REGION Network 3: Обработка аварии по входу №0 / Input 0
   LAB1:
   IF #Input_0 THEN
       #Tmp_Real := #Delay_Sec_0 * 1000.0;
       #Tmp_Time := ROUND(#Tmp_Real);
   END_IF;
   #Timer_0(IN := #Input_0, PT := #Tmp_Time);   // TON
   #_w1 := #Timer_0.Q AND NOT #sarxArrayFlanke[0];   // rising edge
   #sarxArrayFlanke[0] := #Timer_0.Q;
   #sarxArrayMerkers[0] := #_w1;
   #Alarm_0 := (NOT #sarxArrayMerkers[0] AND #Alarm_0) OR (#sarxArrayMerkers[0] AND NOT #Alarm_0);
END_REGION

REGION Network 4: Обработка аварии по входу №1 / Input 1
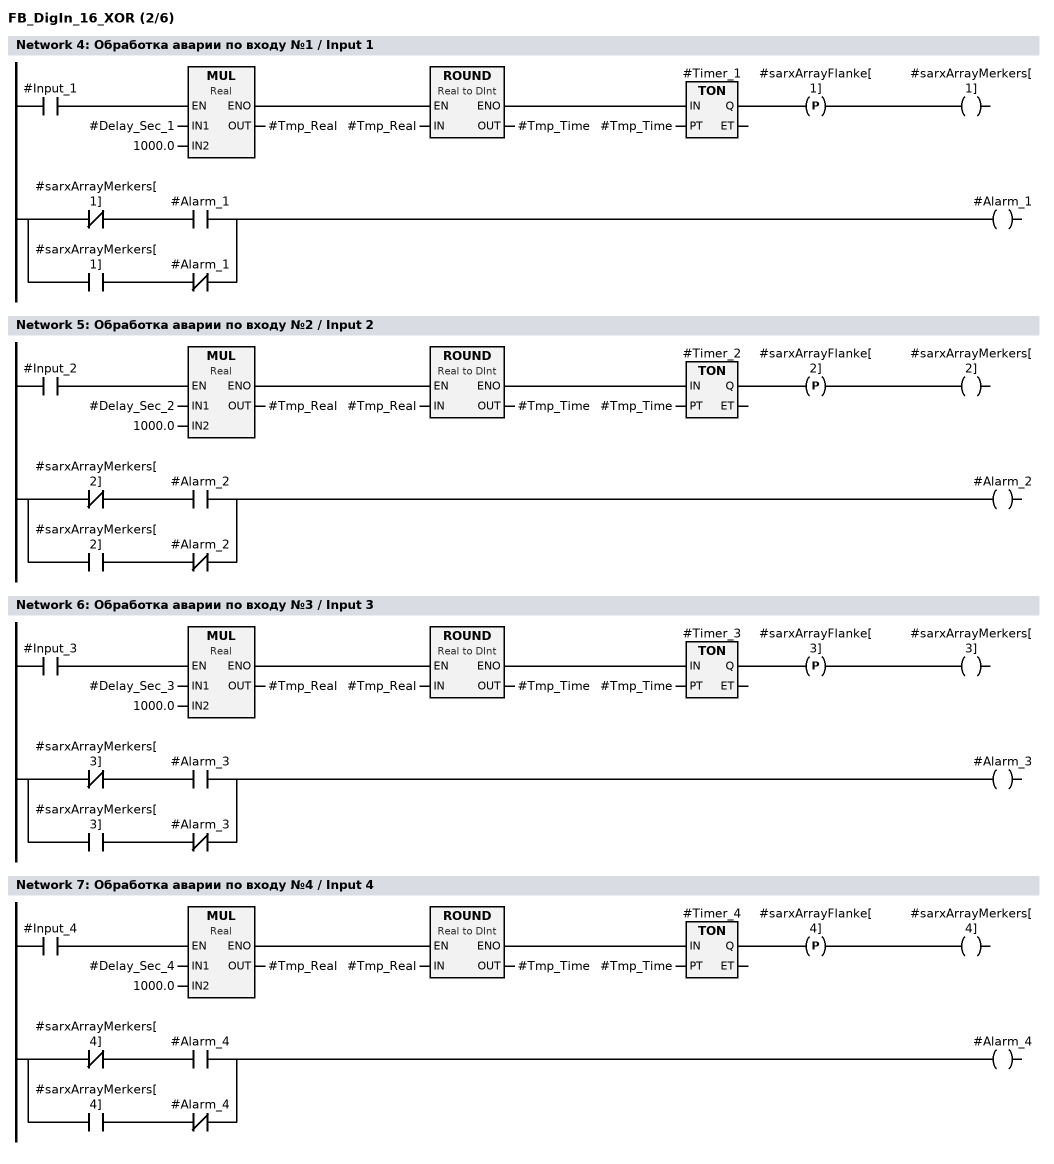
   IF #Input_1 THEN
       #Tmp_Real := #Delay_Sec_1 * 1000.0;
       #Tmp_Time := ROUND(#Tmp_Real);
   END_IF;
   #Timer_1(IN := #Input_1, PT := #Tmp_Time);   // TON
   #_w1 := #Timer_1.Q AND NOT #sarxArrayFlanke[1];   // rising edge
   #sarxArrayFlanke[1] := #Timer_1.Q;
   #sarxArrayMerkers[1] := #_w1;
   #Alarm_1 := (NOT #sarxArrayMerkers[1] AND #Alarm_1) OR (#sarxArrayMerkers[1] AND NOT #Alarm_1);
END_REGION

REGION Network 5: Обработка аварии по входу №2 / Input 2
   IF #Input_2 THEN
       #Tmp_Real := #Delay_Sec_2 * 1000.0;
       #Tmp_Time := ROUND(#Tmp_Real);
   END_IF;
   #Timer_2(IN := #Input_2, PT := #Tmp_Time);   // TON
   #_w1 := #Timer_2.Q AND NOT #sarxArrayFlanke[2];   // rising edge
   #sarxArrayFlanke[2] := #Timer_2.Q;
   #sarxArrayMerkers[2] := #_w1;
   #Alarm_2 := (NOT #sarxArrayMerkers[2] AND #Alarm_2) OR (#sarxArrayMerkers[2] AND NOT #Alarm_2);
END_REGION

REGION Network 6: Обработка аварии по входу №3 / Input 3
   IF #Input_3 THEN
       #Tmp_Real := #Delay_Sec_3 * 1000.0;
       #Tmp_Time := ROUND(#Tmp_Real);
   END_IF;
   #Timer_3(IN := #Input_3, PT := #Tmp_Time);   // TON
   #_w1 := #Timer_3.Q AND NOT #sarxArrayFlanke[3];   // rising edge
   #sarxArrayFlanke[3] := #Timer_3.Q;
   #sarxArrayMerkers[3] := #_w1;
   #Alarm_3 := (NOT #sarxArrayMerkers[3] AND #Alarm_3) OR (#sarxArrayMerkers[3] AND NOT #Alarm_3);
END_REGION

REGION Network 7: Обработка аварии по входу №4 / Input 4
   IF #Input_4 THEN
       #Tmp_Real := #Delay_Sec_4 * 1000.0;
       #Tmp_Time := ROUND(#Tmp_Real);
   END_IF;
   #Timer_4(IN := #Input_4, PT := #Tmp_Time);   // TON
   #_w1 := #Timer_4.Q AND NOT #sarxArrayFlanke[4];   // rising edge
   #sarxArrayFlanke[4] := #Timer_4.Q;
   #sarxArrayMerkers[4] := #_w1;
   #Alarm_4 := (NOT #sarxArrayMerkers[4] AND #Alarm_4) OR (#sarxArrayMerkers[4] AND NOT #Alarm_4);
END_REGION

REGION Network 8: Обработка аварии по входу №5 / Input 5
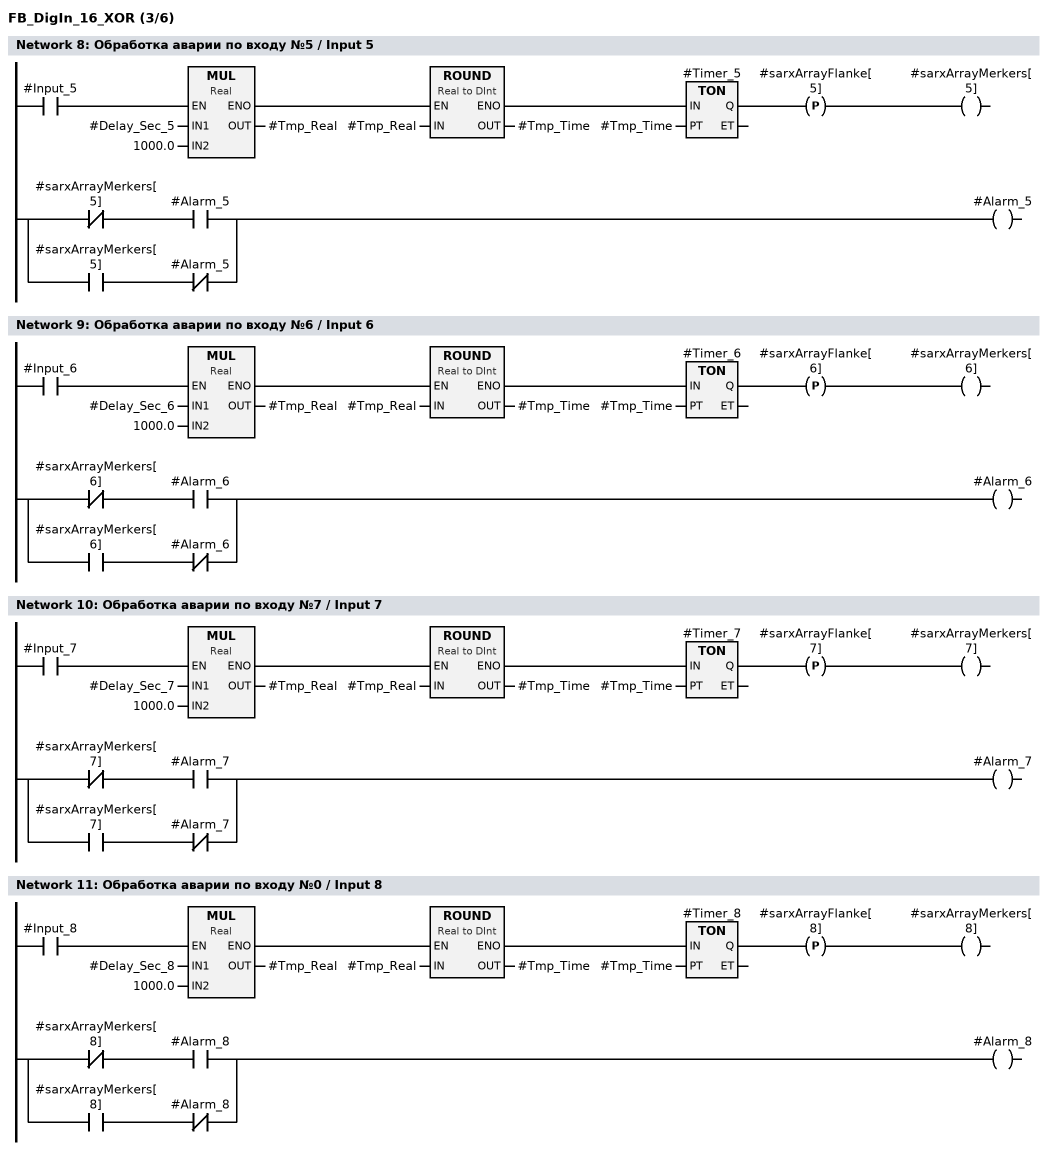
   IF #Input_5 THEN
       #Tmp_Real := #Delay_Sec_5 * 1000.0;
       #Tmp_Time := ROUND(#Tmp_Real);
   END_IF;
   #Timer_5(IN := #Input_5, PT := #Tmp_Time);   // TON
   #_w1 := #Timer_5.Q AND NOT #sarxArrayFlanke[5];   // rising edge
   #sarxArrayFlanke[5] := #Timer_5.Q;
   #sarxArrayMerkers[5] := #_w1;
   #Alarm_5 := (NOT #sarxArrayMerkers[5] AND #Alarm_5) OR (#sarxArrayMerkers[5] AND NOT #Alarm_5);
END_REGION

REGION Network 9: Обработка аварии по входу №6 / Input 6
   IF #Input_6 THEN
       #Tmp_Real := #Delay_Sec_6 * 1000.0;
       #Tmp_Time := ROUND(#Tmp_Real);
   END_IF;
   #Timer_6(IN := #Input_6, PT := #Tmp_Time);   // TON
   #_w1 := #Timer_6.Q AND NOT #sarxArrayFlanke[6];   // rising edge
   #sarxArrayFlanke[6] := #Timer_6.Q;
   #sarxArrayMerkers[6] := #_w1;
   #Alarm_6 := (NOT #sarxArrayMerkers[6] AND #Alarm_6) OR (#sarxArrayMerkers[6] AND NOT #Alarm_6);
END_REGION

REGION Network 10: Обработка аварии по входу №7 / Input 7
   IF #Input_7 THEN
       #Tmp_Real := #Delay_Sec_7 * 1000.0;
       #Tmp_Time := ROUND(#Tmp_Real);
   END_IF;
   #Timer_7(IN := #Input_7, PT := #Tmp_Time);   // TON
   #_w1 := #Timer_7.Q AND NOT #sarxArrayFlanke[7];   // rising edge
   #sarxArrayFlanke[7] := #Timer_7.Q;
   #sarxArrayMerkers[7] := #_w1;
   #Alarm_7 := (NOT #sarxArrayMerkers[7] AND #Alarm_7) OR (#sarxArrayMerkers[7] AND NOT #Alarm_7);
END_REGION

REGION Network 11: Обработка аварии по входу №0 / Input 8
   IF #Input_8 THEN
       #Tmp_Real := #Delay_Sec_8 * 1000.0;
       #Tmp_Time := ROUND(#Tmp_Real);
   END_IF;
   #Timer_8(IN := #Input_8, PT := #Tmp_Time);   // TON
   #_w1 := #Timer_8.Q AND NOT #sarxArrayFlanke[8];   // rising edge
   #sarxArrayFlanke[8] := #Timer_8.Q;
   #sarxArrayMerkers[8] := #_w1;
   #Alarm_8 := (NOT #sarxArrayMerkers[8] AND #Alarm_8) OR (#sarxArrayMerkers[8] AND NOT #Alarm_8);
END_REGION

REGION Network 12: Обработка аварии по входу №0 / Input 9
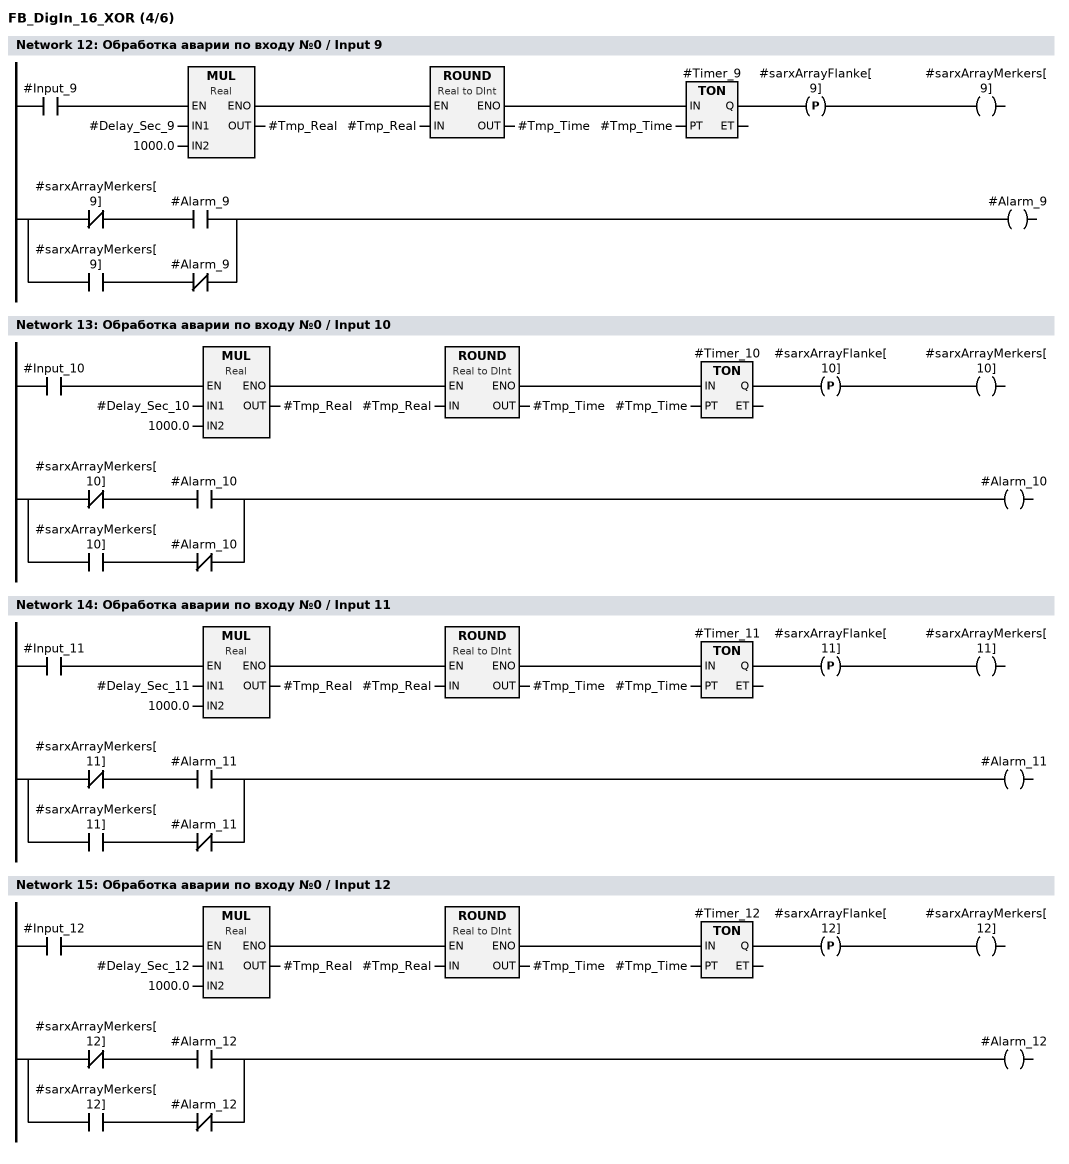
   IF #Input_9 THEN
       #Tmp_Real := #Delay_Sec_9 * 1000.0;
       #Tmp_Time := ROUND(#Tmp_Real);
   END_IF;
   #Timer_9(IN := #Input_9, PT := #Tmp_Time);   // TON
   #_w1 := #Timer_9.Q AND NOT #sarxArrayFlanke[9];   // rising edge
   #sarxArrayFlanke[9] := #Timer_9.Q;
   #sarxArrayMerkers[9] := #_w1;
   #Alarm_9 := (NOT #sarxArrayMerkers[9] AND #Alarm_9) OR (#sarxArrayMerkers[9] AND NOT #Alarm_9);
END_REGION

REGION Network 13: Обработка аварии по входу №0 / Input 10
   IF #Input_10 THEN
       #Tmp_Real := #Delay_Sec_10 * 1000.0;
       #Tmp_Time := ROUND(#Tmp_Real);
   END_IF;
   #Timer_10(IN := #Input_10, PT := #Tmp_Time);   // TON
   #_w1 := #Timer_10.Q AND NOT #sarxArrayFlanke[10];   // rising edge
   #sarxArrayFlanke[10] := #Timer_10.Q;
   #sarxArrayMerkers[10] := #_w1;
   #Alarm_10 := (NOT #sarxArrayMerkers[10] AND #Alarm_10) OR (#sarxArrayMerkers[10] AND NOT #Alarm_10);
END_REGION

REGION Network 14: Обработка аварии по входу №0 / Input 11
   IF #Input_11 THEN
       #Tmp_Real := #Delay_Sec_11 * 1000.0;
       #Tmp_Time := ROUND(#Tmp_Real);
   END_IF;
   #Timer_11(IN := #Input_11, PT := #Tmp_Time);   // TON
   #_w1 := #Timer_11.Q AND NOT #sarxArrayFlanke[11];   // rising edge
   #sarxArrayFlanke[11] := #Timer_11.Q;
   #sarxArrayMerkers[11] := #_w1;
   #Alarm_11 := (NOT #sarxArrayMerkers[11] AND #Alarm_11) OR (#sarxArrayMerkers[11] AND NOT #Alarm_11);
END_REGION

REGION Network 15: Обработка аварии по входу №0 / Input 12
   IF #Input_12 THEN
       #Tmp_Real := #Delay_Sec_12 * 1000.0;
       #Tmp_Time := ROUND(#Tmp_Real);
   END_IF;
   #Timer_12(IN := #Input_12, PT := #Tmp_Time);   // TON
   #_w1 := #Timer_12.Q AND NOT #sarxArrayFlanke[12];   // rising edge
   #sarxArrayFlanke[12] := #Timer_12.Q;
   #sarxArrayMerkers[12] := #_w1;
   #Alarm_12 := (NOT #sarxArrayMerkers[12] AND #Alarm_12) OR (#sarxArrayMerkers[12] AND NOT #Alarm_12);
END_REGION

REGION Network 16: Обработка аварии по входу №0 / Input 13
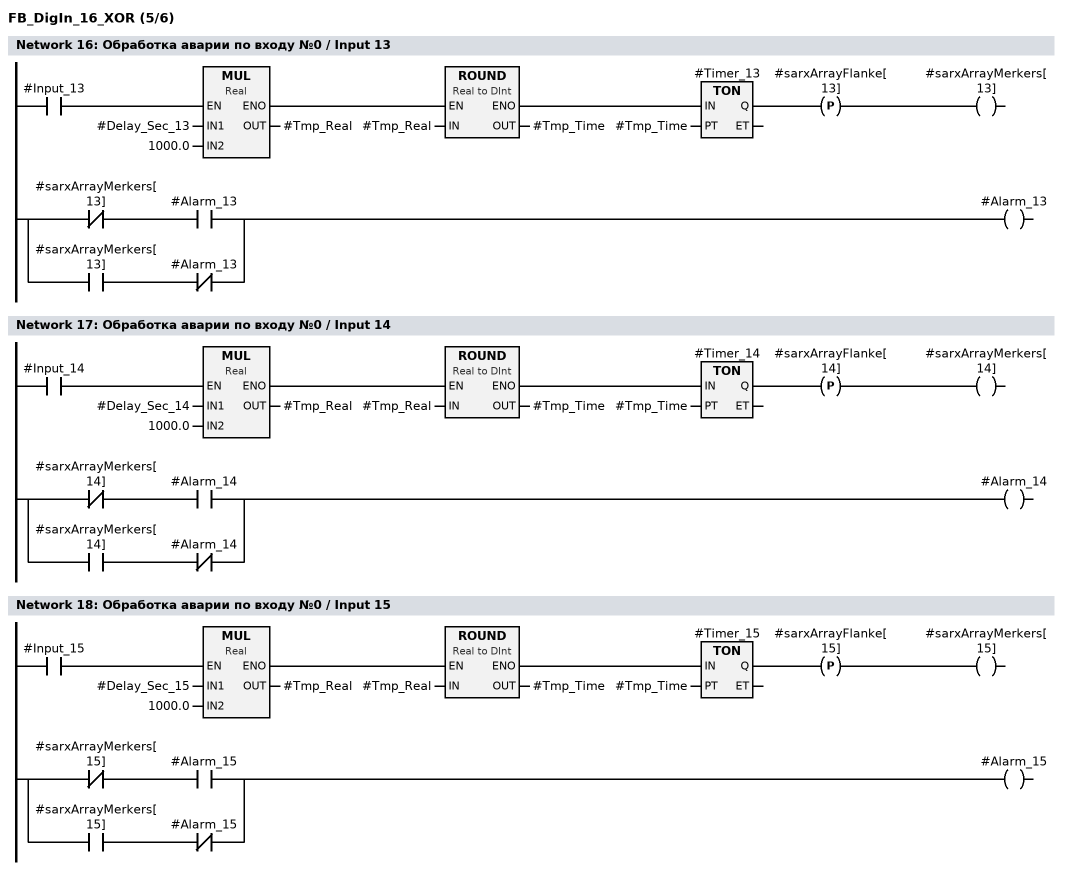
   IF #Input_13 THEN
       #Tmp_Real := #Delay_Sec_13 * 1000.0;
       #Tmp_Time := ROUND(#Tmp_Real);
   END_IF;
   #Timer_13(IN := #Input_13, PT := #Tmp_Time);   // TON
   #_w1 := #Timer_13.Q AND NOT #sarxArrayFlanke[13];   // rising edge
   #sarxArrayFlanke[13] := #Timer_13.Q;
   #sarxArrayMerkers[13] := #_w1;
   #Alarm_13 := (NOT #sarxArrayMerkers[13] AND #Alarm_13) OR (#sarxArrayMerkers[13] AND NOT #Alarm_13);
END_REGION

REGION Network 17: Обработка аварии по входу №0 / Input 14
   IF #Input_14 THEN
       #Tmp_Real := #Delay_Sec_14 * 1000.0;
       #Tmp_Time := ROUND(#Tmp_Real);
   END_IF;
   #Timer_14(IN := #Input_14, PT := #Tmp_Time);   // TON
   #_w1 := #Timer_14.Q AND NOT #sarxArrayFlanke[14];   // rising edge
   #sarxArrayFlanke[14] := #Timer_14.Q;
   #sarxArrayMerkers[14] := #_w1;
   #Alarm_14 := (NOT #sarxArrayMerkers[14] AND #Alarm_14) OR (#sarxArrayMerkers[14] AND NOT #Alarm_14);
END_REGION

REGION Network 18: Обработка аварии по входу №0 / Input 15
   IF #Input_15 THEN
       #Tmp_Real := #Delay_Sec_15 * 1000.0;
       #Tmp_Time := ROUND(#Tmp_Real);
   END_IF;
   #Timer_15(IN := #Input_15, PT := #Tmp_Time);   // TON
   #_w1 := #Timer_15.Q AND NOT #sarxArrayFlanke[15];   // rising edge
   #sarxArrayFlanke[15] := #Timer_15.Q;
   #sarxArrayMerkers[15] := #_w1;
   #Alarm_15 := (NOT #sarxArrayMerkers[15] AND #Alarm_15) OR (#sarxArrayMerkers[15] AND NOT #Alarm_15);
END_REGION

REGION Network 19: Формування статусних слів
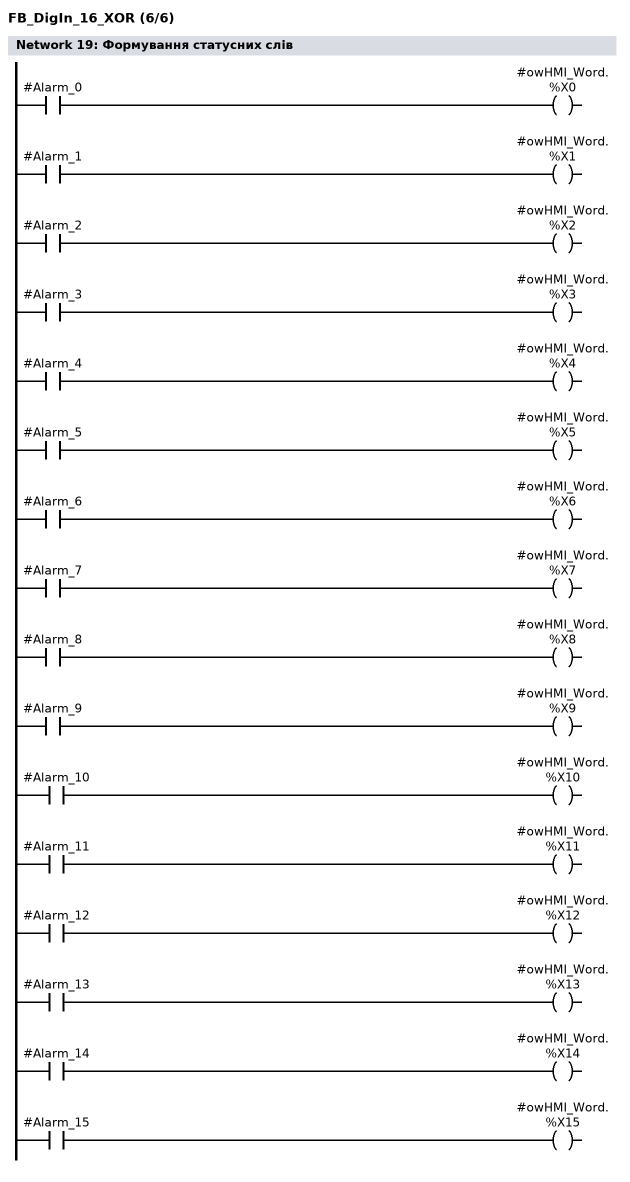
   RUNG wire#powerrail
      Contact( #Alarm_0 )
      Coil( #owHMI_Word.%X0 )
   END_RUNG
   RUNG wire#powerrail
      Contact( #Alarm_1 )
      Coil( #owHMI_Word.%X1 )
   END_RUNG
   RUNG wire#powerrail
      Contact( #Alarm_2 )
      Coil( #owHMI_Word.%X2 )
   END_RUNG
   RUNG wire#powerrail
      Contact( #Alarm_3 )
      Coil( #owHMI_Word.%X3 )
   END_RUNG
   RUNG wire#powerrail
      Contact( #Alarm_4 )
      Coil( #owHMI_Word.%X4 )
   END_RUNG
   RUNG wire#powerrail
      Contact( #Alarm_5 )
      Coil( #owHMI_Word.%X5 )
   END_RUNG
   RUNG wire#powerrail
      Contact( #Alarm_6 )
      Coil( #owHMI_Word.%X6 )
   END_RUNG
   RUNG wire#powerrail
      Contact( #Alarm_7 )
      Coil( #owHMI_Word.%X7 )
   END_RUNG
   RUNG wire#powerrail
      Contact( #Alarm_8 )
      Coil( #owHMI_Word.%X8 )
   END_RUNG
   RUNG wire#powerrail
      Contact( #Alarm_9 )
      Coil( #owHMI_Word.%X9 )
   END_RUNG
   RUNG wire#powerrail
      Contact( #Alarm_10 )
      Coil( #owHMI_Word.%X10 )
   END_RUNG
   RUNG wire#powerrail
      Contact( #Alarm_11 )
      Coil( #owHMI_Word.%X11 )
   END_RUNG
   RUNG wire#powerrail
      Contact( #Alarm_12 )
      Coil( #owHMI_Word.%X12 )
   END_RUNG
   RUNG wire#powerrail
      Contact( #Alarm_13 )
      Coil( #owHMI_Word.%X13 )
   END_RUNG
   RUNG wire#powerrail
      Contact( #Alarm_14 )
      Coil( #owHMI_Word.%X14 )
   END_RUNG
   RUNG wire#powerrail
      Contact( #Alarm_15 )
      Coil( #owHMI_Word.%X15 )
   END_RUNG
   // the same network as SCL:
   #owHMI_Word.%X0 := #Alarm_0;
   #owHMI_Word.%X1 := #Alarm_1;
   #owHMI_Word.%X2 := #Alarm_2;
   #owHMI_Word.%X3 := #Alarm_3;
   #owHMI_Word.%X4 := #Alarm_4;
   #owHMI_Word.%X5 := #Alarm_5;
   #owHMI_Word.%X6 := #Alarm_6;
   #owHMI_Word.%X7 := #Alarm_7;
   #owHMI_Word.%X8 := #Alarm_8;
   #owHMI_Word.%X9 := #Alarm_9;
   #owHMI_Word.%X10 := #Alarm_10;
   #owHMI_Word.%X11 := #Alarm_11;
   #owHMI_Word.%X12 := #Alarm_12;
   #owHMI_Word.%X13 := #Alarm_13;
   #owHMI_Word.%X14 := #Alarm_14;
   #owHMI_Word.%X15 := #Alarm_15;
END_REGION
END_FUNCTION_BLOCK

FUNCTION_BLOCK "FB_StateDefine"   // FB2002, LAD
{ S7_Optimized_Access := 'TRUE' }
VERSION : 0.1
   VAR_INPUT
      irVar : Real;
      irSPVal : Real;
      irGap : Real;
      ixUseNotif : Bool;
      ixUseProcFollow : Bool;
      ixUpDown : Bool;
      ixReset : Bool;
      ixReslease : Bool;
      ixEnControl : Bool;
   END_VAR
   VAR_OUTPUT
      oxLimOK : Bool;
      oxWRN : Bool;
      oxFLT : Bool;
   END_VAR
   VAR
      S1_SR : Bool;
      S2_SR : Bool;
      S3_SR : Bool;
   END_VAR
   VAR_TEMP
      Temp1 : Real;
      Temp2 : Real;
      Temp3 : Bool;
      Temp4 : Bool;
   END_VAR
   VAR_TEMP   // added for the SCL form of the ladder/FBD networks
      _w1 : Bool;
   END_VAR
BEGIN

REGION Network 1
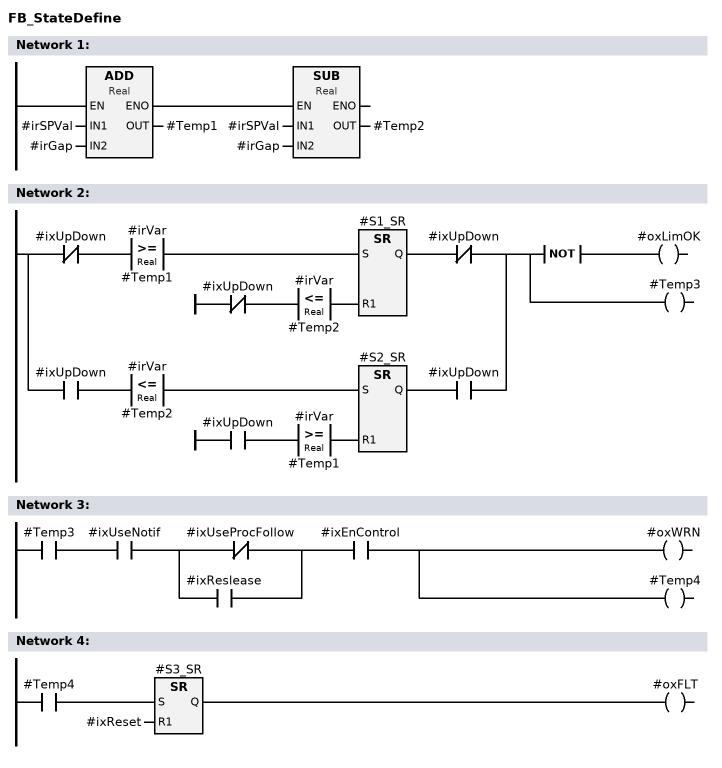
   RUNG wire#powerrail
      { S7_Templates := "SrcType := Real" } Add(in1 := #irSPVal, in2 := #irGap, out => #Temp1)
      { S7_Templates := "SrcType := Real" } Sub(in1 := #irSPVal, in2 := #irGap, out => #Temp2)
   END_RUNG
   // the same network as SCL:
   #Temp1 := #irSPVal + #irGap;
   #Temp2 := #irSPVal - #irGap;
END_REGION

REGION Network 2
   RUNG wire#powerrail
      I_Contact( #ixUpDown )
      { S7_Templates := "SrcType := Real" } GE_Contact(in1 := #irVar, in2 := #Temp1)
      S_SR(operand := #S1_SR, r1 := wire#w1)
      I_Contact( #ixUpDown )
      wire#w2
      Not()
      Coil( #oxLimOK )
   END_RUNG
   RUNG wire#powerrail
      I_Contact( #ixUpDown )
      { S7_Templates := "SrcType := Real" } LE_Contact(in1 := #irVar, in2 := #Temp2)
   END_RUNG wire#w1
   RUNG wire#powerrail
      Contact( #ixUpDown )
      { S7_Templates := "SrcType := Real" } LE_Contact(in1 := #irVar, in2 := #Temp2)
      S_SR(operand := #S2_SR, r1 := wire#w3)
      Contact( #ixUpDown )
   END_RUNG wire#w2
   RUNG wire#powerrail
      Contact( #ixUpDown )
      { S7_Templates := "SrcType := Real" } GE_Contact(in1 := #irVar, in2 := #Temp1)
   END_RUNG wire#w3
   RUNG wire#w2
      Coil( #Temp3 )
   END_RUNG
   // the same network as SCL:
   IF NOT #ixUpDown AND (#irVar >= #Temp1) THEN
       #S1_SR := TRUE;   // SR flip-flop
   END_IF;
   IF NOT #ixUpDown AND (#irVar <= #Temp2) THEN #S1_SR := FALSE; END_IF;
   IF #ixUpDown AND (#irVar <= #Temp2) THEN
       #S2_SR := TRUE;   // SR flip-flop
   END_IF;
   IF #ixUpDown AND (#irVar >= #Temp1) THEN #S2_SR := FALSE; END_IF;
   #_w1 := (#S1_SR AND NOT #ixUpDown) OR (#S2_SR AND #ixUpDown);
   #oxLimOK := NOT #_w1;
   #Temp3 := #_w1;
END_REGION

REGION Network 3
   RUNG wire#powerrail
      Contact( #Temp3 )
      Contact( #ixUseNotif )
      wire#w1
      I_Contact( #ixUseProcFollow )
      wire#w2
      Contact( #ixEnControl )
      wire#w3
      Coil( #oxWRN )
   END_RUNG
   RUNG wire#w1
      Contact( #ixReslease )
   END_RUNG wire#w2
   RUNG wire#w3
      Coil( #Temp4 )
   END_RUNG
   // the same network as SCL:
   #oxWRN := #Temp3 AND #ixUseNotif AND (NOT #ixUseProcFollow OR #ixReslease) AND #ixEnControl;
   #Temp4 := #oxWRN;
END_REGION

REGION Network 4
   RUNG wire#powerrail
      Contact( #Temp4 )
      S_SR(operand := #S3_SR, r1 := #ixReset)
      Coil( #oxFLT )
   END_RUNG
   // the same network as SCL:
   IF #Temp4 THEN
       #S3_SR := TRUE;   // SR flip-flop
   END_IF;
   IF #ixReset THEN #S3_SR := FALSE; END_IF;
   #oxFLT := #S3_SR;
END_REGION
END_FUNCTION_BLOCK

FUNCTION_BLOCK "FB_Bell"   // FB2003, SCL
{ S7_Optimized_Access := 'TRUE' }
VERSION : 0.1
   VAR_INPUT
      ix_9SB1_Bell_Cmd : Bool;   // Сигнал включення дзвінка від оператора
      ix_MechanismsActive : Bool;   // Зафіксовано рух механізмів
   END_VAR
   VAR_OUTPUT
      qx_9K1_Bell_Output : Bool;   // Вихідний сигнал на проміжне реле дзвінка 9К1
   END_VAR
   VAR
      Bell_On_TP : TP_TIME;   // Таймер формування імпульсу тривалістю 1 секунда
      stat_Trigger : R_TRIG;
   END_VAR
BEGIN
   //  ЛОГІКА ЦИКЛІЧНОГО ВМИКАННЯ ДЗВІНКА ГУЧНОГО БОЮ (9К1)
   // А) Виділяємо момент появи сигналу (передній фронт)
   #stat_Trigger(CLK := #ix_MechanismsActive);

   // Б) Запускаємо таймер на 1 секунду в момент появи рух

   #Bell_On_TP(IN:=#stat_Trigger.Q,
               PT:=T#1s);

   // В) Кінцевий вихід на реле дзвінка 9К1 

   #"qx_9K1_Bell_Output" := #"ix_9SB1_Bell_Cmd" OR #Bell_On_TP.Q;
END_FUNCTION_BLOCK

FUNCTION_BLOCK "FB_DIAG_SCALANCE"   // FB2004, SCL
{ S7_Optimized_Access := 'TRUE' }
VERSION : 1.0
   VAR_INPUT
      HW_DEVICE : Hw_Device;
      HW_IO : Hw_Io;
   END_VAR
   VAR_OUTPUT
      NodeOk : Bool;
      NodeFlt : Bool;
      RingOk : Bool;
      DiagnosticsValid : Bool;
      RingStateValid : Bool;
   END_VAR
   VAR
      Node : "FB_DIAG_NODE";
   END_VAR
BEGIN

       #Node(HW_DEVICE := #HW_DEVICE);
       #NodeOk := #Node.ModulesOk;
       #NodeFlt := #Node.ModulesFlt;
       #DiagnosticsValid := #Node.DiagnosticsValid;
       // The SCALANCE is an MRP client. Use the CPU manager's validated state.
       // Published by FC_MRP_Publish later in the same cyclic diagnostic call.
       #RingStateValid := "DB_Diag_Prof".Ring_StateValid;
       #RingOk := #RingStateValid AND "DB_Diag_Prof".Ring_Ok;
END_FUNCTION_BLOCK

FUNCTION_BLOCK "FB_DIAG_NODE"   // FB2005, SCL
{ S7_Optimized_Access := 'TRUE' }
VERSION : 1.0
   VAR_INPUT
      HW_DEVICE : Hw_Device;
   END_VAR
   VAR_OUTPUT
      NodeOk : Bool;
      NodeFlt : Bool;
      ModulesOk : Bool;
      ModulesFlt : Bool;
      PresenceValid : Bool;
      FaultsValid : Bool;
      DiagnosticsValid : Bool;
      PresenceStatus : Int;
      FaultStatus : Int;   // Lower bound -1 maps the summary bit to -1 and module slot n to [n].
   END_VAR
   VAR
      MODULES_EXISTS : Array[-1..126] of Bool;
      MODULES_FLT : Array[-1..126] of Bool;
   END_VAR
   VAR_TEMP
      i : Int;
   END_VAR
BEGIN

       #PresenceStatus := ModuleStates(LADDR := #HW_DEVICE, MODE := 4, STATE := #MODULES_EXISTS);
       #FaultStatus := ModuleStates(LADDR := #HW_DEVICE, MODE := 2, STATE := #MODULES_FLT);
       #PresenceValid := #PresenceStatus = 0;
       #FaultsValid := #FaultStatus = 0;
       #DiagnosticsValid := #PresenceValid AND #FaultsValid;
       // Invalid reads cannot leave old module data appearing healthy.
       IF NOT #PresenceValid THEN
           FOR #i := -1 TO 126 DO #MODULES_EXISTS[#i] := FALSE; END_FOR;
       END_IF;
       IF NOT #FaultsValid THEN
           FOR #i := -1 TO 126 DO #MODULES_FLT[#i] := TRUE; END_FOR;
       END_IF;
       #NodeOk := #PresenceValid AND #MODULES_EXISTS[-1];
       #NodeFlt := NOT #NodeOk;
       #ModulesOk := #NodeOk AND #FaultsValid AND NOT #MODULES_FLT[-1];
       // Existing machine permissives fail closed on unavailable diagnostics.
       // DiagnosticsValid distinguishes unavailable data from a confirmed fault.
       #ModulesFlt := NOT #ModulesOk;
END_FUNCTION_BLOCK

FUNCTION "FC_Filter" : Void   // FC2000, SCL
{ S7_Optimized_Access := 'TRUE' }
VERSION : 0.1
   VAR_INPUT
      irVal : Real;
      iiFTime : Int;
   END_VAR
   VAR_OUTPUT
      orVal : Real;
   END_VAR
   VAR_TEMP
      CycleNumber : Real;
      cA : Real;
      cB : Real;
      FVal : Real;
      FVal_Old : Real;
   END_VAR
BEGIN
   #CycleNumber := (INT_TO_REAL(#iiFTime) * 0.1);
   #cA := #CycleNumber / (#CycleNumber + 1.0);
   #cB := 1.0 / (#CycleNumber + 1.0);
   #FVal := #cB * #irVal + #cA * #FVal_Old;
   #FVal_Old := #FVal;
   #orVal := #FVal;
END_FUNCTION

FUNCTION "FC_Rem_Ctrl" : Void   // FC2001, LAD
{ S7_Optimized_Access := 'TRUE' }
VERSION : 0.1
   VAR_INPUT
      RemCtrl_IN : "udtRemCtrl";
   END_VAR
   VAR_OUTPUT
      RemCtrl_OUT : "udtRemCtrl";
   END_VAR
BEGIN

REGION Network 1: 1SB1 Підйом 1 швидкість
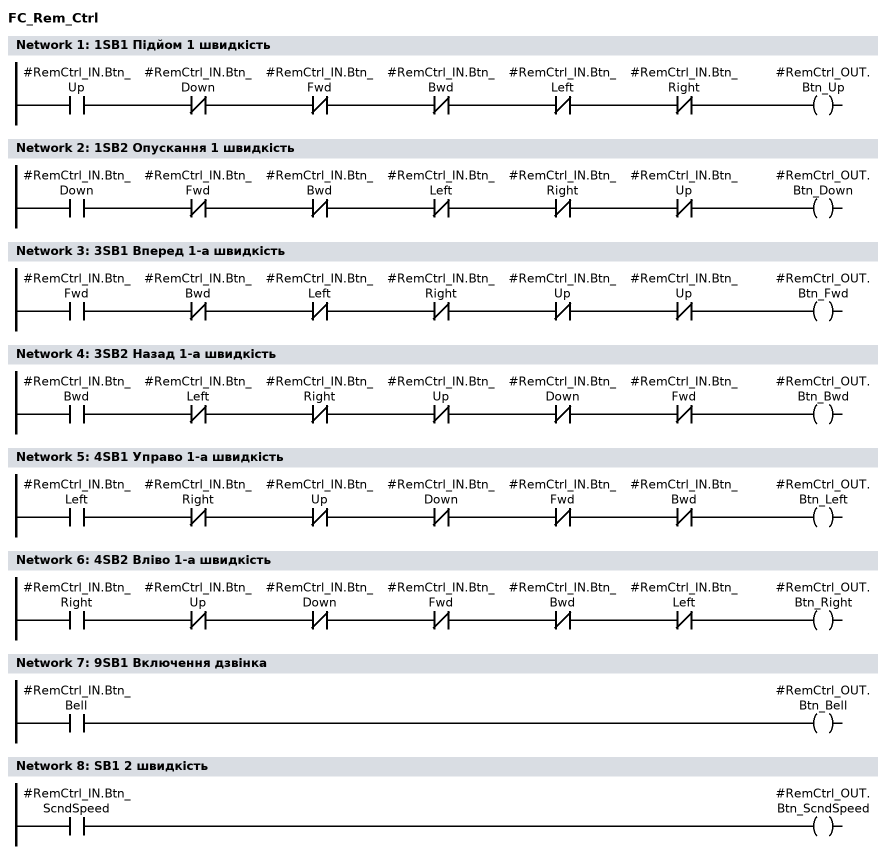
   RUNG wire#powerrail
      Contact( #RemCtrl_IN.Btn_Up )
      I_Contact( #RemCtrl_IN.Btn_Down )
      I_Contact( #RemCtrl_IN.Btn_Fwd )
      I_Contact( #RemCtrl_IN.Btn_Bwd )
      I_Contact( #RemCtrl_IN.Btn_Left )
      I_Contact( #RemCtrl_IN.Btn_Right )
      Coil( #RemCtrl_OUT.Btn_Up )
   END_RUNG
   // the same network as SCL:
   #RemCtrl_OUT.Btn_Up := #RemCtrl_IN.Btn_Up AND NOT #RemCtrl_IN.Btn_Down AND NOT #RemCtrl_IN.Btn_Fwd AND NOT #RemCtrl_IN.Btn_Bwd AND NOT #RemCtrl_IN.Btn_Left AND NOT #RemCtrl_IN.Btn_Right;
END_REGION

REGION Network 2: 1SB2 Опускання 1 швидкість
   RUNG wire#powerrail
      Contact( #RemCtrl_IN.Btn_Down )
      I_Contact( #RemCtrl_IN.Btn_Fwd )
      I_Contact( #RemCtrl_IN.Btn_Bwd )
      I_Contact( #RemCtrl_IN.Btn_Left )
      I_Contact( #RemCtrl_IN.Btn_Right )
      I_Contact( #RemCtrl_IN.Btn_Up )
      Coil( #RemCtrl_OUT.Btn_Down )
   END_RUNG
   // the same network as SCL:
   #RemCtrl_OUT.Btn_Down := #RemCtrl_IN.Btn_Down AND NOT #RemCtrl_IN.Btn_Fwd AND NOT #RemCtrl_IN.Btn_Bwd AND NOT #RemCtrl_IN.Btn_Left AND NOT #RemCtrl_IN.Btn_Right AND NOT #RemCtrl_IN.Btn_Up;
END_REGION

REGION Network 3: 3SB1 Вперед 1-а швидкість
   RUNG wire#powerrail
      Contact( #RemCtrl_IN.Btn_Fwd )
      I_Contact( #RemCtrl_IN.Btn_Bwd )
      I_Contact( #RemCtrl_IN.Btn_Left )
      I_Contact( #RemCtrl_IN.Btn_Right )
      I_Contact( #RemCtrl_IN.Btn_Up )
      I_Contact( #RemCtrl_IN.Btn_Up )
      Coil( #RemCtrl_OUT.Btn_Fwd )
   END_RUNG
   // the same network as SCL:
   #RemCtrl_OUT.Btn_Fwd := #RemCtrl_IN.Btn_Fwd AND NOT #RemCtrl_IN.Btn_Bwd AND NOT #RemCtrl_IN.Btn_Left AND NOT #RemCtrl_IN.Btn_Right AND NOT #RemCtrl_IN.Btn_Up AND NOT #RemCtrl_IN.Btn_Up;
END_REGION

REGION Network 4: 3SB2 Назад 1-а швидкість
   RUNG wire#powerrail
      Contact( #RemCtrl_IN.Btn_Bwd )
      I_Contact( #RemCtrl_IN.Btn_Left )
      I_Contact( #RemCtrl_IN.Btn_Right )
      I_Contact( #RemCtrl_IN.Btn_Up )
      I_Contact( #RemCtrl_IN.Btn_Down )
      I_Contact( #RemCtrl_IN.Btn_Fwd )
      Coil( #RemCtrl_OUT.Btn_Bwd )
   END_RUNG
   // the same network as SCL:
   #RemCtrl_OUT.Btn_Bwd := #RemCtrl_IN.Btn_Bwd AND NOT #RemCtrl_IN.Btn_Left AND NOT #RemCtrl_IN.Btn_Right AND NOT #RemCtrl_IN.Btn_Up AND NOT #RemCtrl_IN.Btn_Down AND NOT #RemCtrl_IN.Btn_Fwd;
END_REGION

REGION Network 5: 4SB1 Управо 1-а швидкість
   RUNG wire#powerrail
      Contact( #RemCtrl_IN.Btn_Left )
      I_Contact( #RemCtrl_IN.Btn_Right )
      I_Contact( #RemCtrl_IN.Btn_Up )
      I_Contact( #RemCtrl_IN.Btn_Down )
      I_Contact( #RemCtrl_IN.Btn_Fwd )
      I_Contact( #RemCtrl_IN.Btn_Bwd )
      Coil( #RemCtrl_OUT.Btn_Left )
   END_RUNG
   // the same network as SCL:
   #RemCtrl_OUT.Btn_Left := #RemCtrl_IN.Btn_Left AND NOT #RemCtrl_IN.Btn_Right AND NOT #RemCtrl_IN.Btn_Up AND NOT #RemCtrl_IN.Btn_Down AND NOT #RemCtrl_IN.Btn_Fwd AND NOT #RemCtrl_IN.Btn_Bwd;
END_REGION

REGION Network 6: 4SB2 Вліво 1-а швидкість
   RUNG wire#powerrail
      Contact( #RemCtrl_IN.Btn_Right )
      I_Contact( #RemCtrl_IN.Btn_Up )
      I_Contact( #RemCtrl_IN.Btn_Down )
      I_Contact( #RemCtrl_IN.Btn_Fwd )
      I_Contact( #RemCtrl_IN.Btn_Bwd )
      I_Contact( #RemCtrl_IN.Btn_Left )
      Coil( #RemCtrl_OUT.Btn_Right )
   END_RUNG
   // the same network as SCL:
   #RemCtrl_OUT.Btn_Right := #RemCtrl_IN.Btn_Right AND NOT #RemCtrl_IN.Btn_Up AND NOT #RemCtrl_IN.Btn_Down AND NOT #RemCtrl_IN.Btn_Fwd AND NOT #RemCtrl_IN.Btn_Bwd AND NOT #RemCtrl_IN.Btn_Left;
END_REGION

REGION Network 7: 9SB1 Включення дзвінка
   RUNG wire#powerrail
      Contact( #RemCtrl_IN.Btn_Bell )
      Coil( #RemCtrl_OUT.Btn_Bell )
   END_RUNG
   // the same network as SCL:
   #RemCtrl_OUT.Btn_Bell := #RemCtrl_IN.Btn_Bell;
END_REGION

REGION Network 8: SB1 2 швидкість
   RUNG wire#powerrail
      Contact( #RemCtrl_IN.Btn_ScndSpeed )
      Coil( #RemCtrl_OUT.Btn_ScndSpeed )
   END_RUNG
   // the same network as SCL:
   #RemCtrl_OUT.Btn_ScndSpeed := #RemCtrl_IN.Btn_ScndSpeed;
END_REGION
END_FUNCTION

FUNCTION "FC_ARRAY_LEN" : Int   // FC2002, SCL
TITLE = Array length (amount of elements)
{ S7_Optimized_Access := 'FALSE' }
AUTHOR : PIA
FAMILY : Array
VERSION : 0.1
// DANIELI AUTOMATION S.p.A.
// Flat Products Department
// 
// This block manages:
// Array length
// 
// Revisions history:
// 01 - 22/06/2015 - Issue TIA Portal - PIA user
// 
// This software is sold with the expressed agreement that the information therein
// contained is the property of DANIELI AUTOMATION S.p.A. It will not be
// reproduced, installed, copied or otherwise disposed or directly or indirectly
// for different uses than the scope of this contract, and will not be used, in
// whole or in part, to assist in making or to furnish information for the use of
// the software, or other reproductions hereof, or for the making of software or
// parts thereof, except upon written permission of DANIELI AUTOMATION S.p.A.
// obtained and specific to each case. The acceptance of this software will be
// constructed as an acceptance of the foregoing agreement.
   VAR_INPUT
      src : Variant;   // Array
   END_VAR
   // Ret_Val : Amount of array elements
BEGIN
   //return amount of array elements 
   IF IS_ARRAY(#src) THEN
       ENO := 1;
       #FC_ARRAY_LEN := UDINT_TO_INT(CountOfElements(#src));
   ELSE
       ENO := 0;
       #FC_ARRAY_LEN := -1;
   END_IF;
END_FUNCTION

// folder: 20_PSM

FUNCTION_BLOCK "FB_PSM_LC"   // FB20, SCL
{ S7_Optimized_Access := 'TRUE' }
VERSION : 0.1
// Лінійний контактор
   VAR_INPUT
      ix_6SF1_Breaker_6KV : Bool;   // Вимикач живлення 6KV
      ix_6KV_VoltageCtrl_380V : Bool;   // Контроль напруги введення 380В
      ix_6SF5_HeaterBreaker : Bool;   // Вимикач кіл живлення обігріву
      ix_6QF2_BrakeCircuitProt : Bool;   // Захист кіл гальм
      ix_6QF3_TransfBreaker_6T1 : Bool;   // Вимикач трансформатора 6T1
      ix_6QF4_TransfSecBreaker : Bool;   // Вимикач вторинних кіл трансформатора 6T1
      ix_6SF2_CtrlCircuit_220V : Bool;   // Вимикач кіл управління 220В
      ix_6SF4_OVP_Power_220V : Bool;   // Вимикач кіл живлення ОВП 220В
      ix_9QF4_CabinetAux_220V : Bool;   // Вимикач власних потреб шафи 220В
      ix_9K2_CabinetHeating : Bool;   // Контроль підігріву шафи (необхідний тільки при старті)
      ix_1QF1_BrakeRectifier_1YB1 : Bool;   // Захист випрямляча гальма 1YB1
      ix_1QF2_BrakeRectifier_1YB2 : Bool;   // Захист випрямляча гальма 1YB2
      ix_4QF1_BrakeCircuitProt : Bool;   // Захист кіл гальм
      ix_K3_SeismicAlarm : Bool;   // Сигнал сейсмодатчика
      ix_Profinet_OK : Bool;   // Статус комунікації Profinet
      ix_FireAlarm : Bool;   // Пожежна тривога
      ix_6K3_CmdStart : Bool;   // 6К3 Команда на включение лінійного контактора з пульта
      ix_6KM1_Feedback_LC : Bool;   // 6KM1 Лінійний контактор включений
      ix_6KM2_Feedback_Ctrl220 : Bool;   // 6KM2 Контактор кіл керування 220в включений
      is_MovePerm : "udtMovePerm";   // Кінцеві вимикачі руху крайніх положень
      is_Manual_interlock : "udtMDM";   // Дозволи роботи механізмів (РП роз'єднано / ручний привід відсутній)
      is_RemCtrl : "udtRemCtrl";   // Кнопки руху з пульта (для контролю нульового положення при старті)
      is_SpeedPerm : "udtSpeedPerm";   // Дозвіл ном. швидкості
      ix_Ack : Bool;   // Сигнал квітування помилок з панелі
   END_VAR
   VAR_OUTPUT
      qx_6K1_Permit_LC : Bool;   // 6K1 Дозвіл включення лінійного контактора
      qx_6K2_Hold_LC : Bool;   // 6K2 Вимкнення лінійного контактора (коло утримання)
      qx_6HL1_SignalStart : Bool;   // 6HL1 Сигналізація про запуск контактора
      qx_6HL2_SignalVoltage : Bool;   // 6HL2 Сигналізація про стан вхідної напруги
      qx_Zero_Protection_Active : Bool;   // Активовано блокування «Нульовий захист» (затиснуті кнопки)
      qx_Alarm_Active : Bool;   // Загальний прапор критичної аварії контактора
      qw_Alarm_Code : Word;   // Код помилки для панелі ЛМІ
      qw_Trip_1 : Word;   // Слово 1 фіксації причин відключення
      qw_Trip_2 : Word;   // Слово 2 фіксації причин відключення
   END_VAR
   VAR
      stat_InterlockStartup : Bool;   // Прапор захисту від старту при натиснутих органах керування
      stat_Prev_KM1_Feedback : Bool;   // Прапор для відстеження моменту відключення контактора END_VAREND_INTERFACEИспользуйте код с осторожностью.💻 Оновлений код програми на мові SCLscl// =========================================================================================// ЛОГІКА КЕРУВАННЯ ЛІНІЙНИМ КОНТАКТОРОМ (ЛК) З ФІКСАЦІЄЮ ПРИЧИНИ ВІДКЛЮЧЕННЯ// Категорія функції за НП 306.2.202-2015: В (Програмний технологічний захисний блок)// =========================================================================================//------------------------------------------------------------------------------------------// ЗБІР ЗАГАЛЬНИХ УМОВ УВІМКНЕННЯ ТА РОБОТИ (Пункт 1, Сторінка 13 ТЗ)//------------------------------------------------------------------------------------------#q_HL2_SignalVoltage := #i_SF1_Breaker_6KV AND #i_KV_VoltageCtrl_380V; // Сигналізація вхідної напруги// Базові апаратні умови готовності електрообладнання#stat_LC_Active := #i_SF1_Breaker_6KV AND #i_KV_VoltageCtrl_380V AND #i_SF5_HeaterBreaker AND #i_QF2_BrakeCircuitProt AND #i_QF3_TransfBreaker_6T1 AND #i_QF4_TransfSecBreaker AND #i_SF2_CtrlCircuit_220V AND #i_SF4_OVP_Power_220V AND #i_QF4_CabinetAux_220V AND #i_QF1_BrakeRectifier_1YB1 AND #i_QF2_BrakeRectifier_1YB2 AND #i_QF1_BrakeCircuitProt_4;// Перевірка дозволів роботи механізмів (ручні привода відключені / РП роз'єднані)#stat_LC_Active := #stat_LC_Active AND #i_SQ33_Brake_1YB2_OK AND #i_SQ41_HoistManual_OK AND #i_SQ41_TrolleyManual_OK AND #i_SQ41_GantryManual1_OK AND #i_SQ42_GantryManual2_OK;// Контроль кінцевих вимикачів руху крайніх положень (Пункт 1.15 та Пункт 8)#stat_LC_Active := #stat_LC_Active AND #i_K4_GantryRight_Limit AND #i_K3_GantryLeft_Limit AND #i_K4_HoistDown_Limit AND #i_K3_HoistUp_Limit AND #i_K4_TrolleyBackward_Limit AND #i_K2_TrolleyForward_Limit;// Інтеграція умов щодо сейсміки та мережі Profinet#stat_LC_Active := #stat_LC_Active AND NOT #i_K3_SeismicAlarm AND #i_Profinet_OK;//------------------------------------------------------------------------------------------// ЗАХИСТ ВІД НЕСАНКЦІОНОВАНОГО ПУСКУ (Нульовий захист)//------------------------------------------------------------------------------------------IF NOT #i_K3_CmdStart AND NOT #i_Btn_HoistUp AND NOT #i_Btn_HoistDown AND NOT #i_Btn_TrolleyFwd AND NOT #i_Btn_TrolleyBwd AND NOT #i_Btn_GantryLeft AND NOT #i_Btn_GantryRight THEN #stat_InterlockStartup := FALSE; END_IF;IF (#stat_LC_Active AND NOT #q_K2_Hold_LC AND #i_K3_CmdStart) AND NOT #stat_InterlockStartup THEN IF NOT #i_K2_CabinetHeating THEN #stat_InterlockStartup := TRUE; END_IF;END_IF;//------------------------------------------------------------------------------------------// ПРОЦЕДУРА УВІМКНЕННЯ ТА СТРУКТУРА УДЕРЖАННЯ (Сторінка 14 ТЗ)//------------------------------------------------------------------------------------------IF #stat_LC_Active AND #i_K2_CabinetHeating AND NOT #stat_InterlockStartup AND (#stat_AlarmReg = 16#0000) THEN IF #i_K3_CmdStart THEN #q_K2_Hold_LC := TRUE; IF NOT #i_KM1_Feedback_LC THEN #q_K1_Permit_LC := TRUE; END_IF; END_IF;ELSE // Умови вимкнення контактора (Пункт 2, Сторінка 14) #q_K2_Hold_LC := FALSE; #q_K1_Permit_LC := FALSE; END_IF;IF #i_KM1_Feedback_LC THEN #q_K1_Permit_LC := FALSE;END_IF;IF NOT #q_K2_Hold_LC THEN #q_K1_Permit_LC := FALSE;END_IF;#q_HL1_SignalStart := #i_KM1_Feedback_LC;//------------------------------------------------------------------------------------------// КОНТРОЛЬ ЗАХИСТІВ ТА ДІАГНОСТИКА АВАРІЙНИХ ПОДІЙ//------------------------------------------------------------------------------------------#stat_TimerFeedback(IN := #q_K1_Permit_LC AND NOT #i_KM1_Feedback_LC, PT := T#2s);// Наповнення динамічного регістру помилокIF #stat_TimerFeedback.Q THEN #stat_AlarmReg.%X0 := TRUE; // Бит 0: Аварія часу очікування замикання контактора 6KM1END_IF;IF #i_KM1_Feedback_LC AND NOT #i_KM2_Feedback_Ctrl220 THEN #stat_AlarmReg.%X1 := TRUE; // Бит 1: Відсутність або зникнення сигналу 6КМ2 #q_K2_Hold_LC := FALSE; END_IF;IF NOT #q_K2_Hold_LC AND #i_KM1_Feedback_LC THEN #stat_AlarmReg.%X2 := TRUE; // Бит 2: Спонтанне замикання контактора без командиEND_IF;IF NOT #stat_LC_Active AND #i_KM1_Feedback_LC THEN #stat_AlarmReg.%X3 := TRUE; // Бит 3: Спрацювання загальних блокувань/кінцевиків під час роботиEND_IF;//------------------------------------------------------------------------------------------// ФІКСАЦІЯ КОНКРЕТНОЇ ПРИЧИНИ ТРИГЕРУ ВІДКЛЮЧЕННЯ (НОВИЙ БЛОК ЛОГІКИ)//------------------------------------------------------------------------------------------// Ловимо задній фронт сигналу зворотного зв'язку контактора (момент розмикання 6KM1)IF #stat_Prev_KM1_Feedback AND NOT #i_KM1_Feedback_LC THEN // Обнуляємо попереднє значення перед записом нового трипу #q_Trip_Reason_Code := 16#0000; // Аналізуємо побітово, яка саме причина призвела до відключення в цей момент: // Група внутрішнього контролю таймінгів та колізій #q_Trip_Reason_Code.%X0 := #stat_AlarmReg.%X0; // Аварія таймауту включення 6KM1 #q_Trip_Reason_Code.%X1 := NOT #i_KM2_Feedback_Ctrl220; // Зникнення або відсутність 6КМ2 (цепі 220В) // Група автоматів живлення та захисту (Пункт 1) #q_Trip_Reason_Code.%X2 := NOT #i_SF1_Breaker_6KV OR NOT #i_KV_VoltageCtrl_380V; // Проблема з головним вводом #q_Trip_Reason_Code.%X3 := NOT #i_SF2_CtrlCircuit_220V OR NOT #i_SF4_OVP_Power_220V; // Вимкнено автомати кіл керування #q_Trip_Reason_Code.%X4 := NOT #i_QF3_TransfBreaker_6T1 OR NOT #i_QF4_TransfSecBreaker; // Проблема з трансформатором 6Т1 #q_Trip_Reason_Code.%X5 := NOT #i_QF2_BrakeCircuitProt OR NOT #i_QF1_BrakeCircuitProt_4; // Автомати захисту кіл гальм #q_Trip_Reason_Code.%X6 := NOT #i_QF1_BrakeRectifier_1YB1 OR NOT #i_QF2_BrakeRectifier_1YB2; // Випрямлячі гальм // Група дозволів та безпеки механізмів #q_Trip_Reason_Code.%X7 := NOT #i_SQ41_HoistManual_OK OR NOT #i_SQ33_Brake_1YB2_OK; // Ручний привід або гальмо підйому не в нормі #q_Trip_Reason_Code.%X8 := NOT #i_SQ41_TrolleyManual_OK; // РП візка не роз'єднано #q_Trip_Reason_Code.%X9 := NOT #i_SQ41_GantryManual1_OK OR NOT #i_SQ42_GantryManual2_OK; // РП моста не роз'єднано // Кінцеві вимикачі крайніх положень (Пункт 8 ТЗ) #q_Trip_Reason_Code.%X10 := NOT #i_K3_HoistUp_Limit OR NOT #i_K4_HoistDown_Limit; // Спрацював кінцевик підйому (верх/низ) #q_Trip_Reason_Code.%X11 := NOT #i_K2_TrolleyForward_Limit OR NOT #i_K4_TrolleyBackward_Limit; // Кінцевик візка (вперед/назад) #q_Trip_Reason_Code.%X12 := NOT #i_K3_GantryLeft_Limit OR NOT #i_K4_GantryRight_Limit; // Кінцевик моста (ліво/право) // Зовнішні критичні фактори #q_Trip_Reason_Code.%X13 := #i_K3_SeismicAlarm; // Сейсмічна активність (аварія) #q_Trip_Reason_Code.%X14 := NOT #i_Profinet_OK; // Втрата зв'язку по Profinet // Якщо жоден із захистів вище не зафіксовано, але контактор відключився — це було ручне відключення оператором (або кнопка Стоп) IF #q_Trip_Reason_Code = 16#0000 THEN #q_Trip_Reason_Code.%X15 := TRUE; // Нормальне технологічне вимкнення оператором END_IF;END_IF;// Зберігаємо поточний стан для наступного циклу PLC#stat_Prev_KM1_Feedback := #i_KM1_Feedback_LC;//------------------------------------------------------------------------------------------// КВІТУВАННЯ ТА СКИДАННЯ ПОМИЛОК//------------------------------------------------------------------------------------------IF #i_Ack THEN #stat_AlarmReg := 16#0000; #stat_InterlockStartup := FALSE; // Скидаємо слово причини відключення тільки тоді, коли оператор усвідомлено натиснув квітування #q_Trip_Reason_Code := 16#0000;END_IF;#q_Alarm_Active := (#stat_AlarmReg <> 16#0000);#q_Alarm_Code := #stat_AlarmReg;Используйте код с осторожностью.📋 Карта розшифровки бітів слова q_Trip_Reason_Code для HMI/ЛМИ:Коли на панелі оператора відображається аварія, це слово покаже точну причину (можна налаштувати тригери текстових повідомлень у TIA Portal WinCC):Bit 0 (0x0001) — Контактор 6KM1 не зміг замикатися протягом 2 секунд після команди.Bit 1 (0x0002) — Зник зворотний зв'язок від контактора кіл управління 220В (6KM2).Bit 2 (0x0004) — Пропало живлення 6КВ або є проблеми з реле контролю напруги 380В.Bit 3 (0x0008) — Вимкнено автомати кіл керування SF2 або ОВП SF4.Bit 4 (0x0010) — Аварія автоматів трансформатора 6Т1 (первинна або вторинна обмотка).Bit 5 (0x0020) — Спрацював захист автоматів живлення гальм.Bit 6 (0x0040) — Спрацював захист випрямлячів гальм 1YB1 або 1YB2.Bit 7 (0x0080) — Порушено безпеку підйому (ручний привід не заблоковано або гальмо 1YB2 в аварії).Bit 8 (0x0100) — Ручний привід пересування візка не від'єднано.Bit 9 (0x0200) — Ручний привід пересування моста (приводи 1 або 2) не від'єднано.Bit 10 (0x0400) — Механізм дійшов до аварійного кінцевого вимикача підйому (Верх/Низ).Bit 11 (0x0800) — Механізм дійшов до аварійного кінцевого вимикача візка (Вперед/Назад).Bit 12 (0x1000) — Механізм дійшов до аварійного кінцевого вимикача моста (Ліво/Право).Bit 13 (0x2000) — Спрацював сейсмічний захист крана (датчик 9К3).Bit 14 (0x4000) — Відключення через критичну помилку мережі Profinet.Bit 15 (0x8000) — Нормальне планове вимкнення контактора (команда оператора, без аварій).Тепер діагностика лінійного контактора стала повністю інформативною та відповідає вимогам до кранових систем ядерних установок.Чи є необхідність інтегрувати передачу цього слова по Profinet до вищого рівня АСУ ТП, чи переходимо до розробки логіки наступного кроку — управління гальмами механізму підйому?
      stat_LC_Active : Bool;   // Внутрішній статус готовності до роботи контактора
      stat_AlarmReg : Word;   // Регістр аварійних подій контактора
      stat_TimerFeedback : TON_TIME;   // Таймер контролю часу увімкнення контактора
      stat_TimerFeedback_Con : TON_TIME;   // Таймер контролю часу увімкнення контактора
      stat_TimerFeedback_LC : TON_TIME;   // Таймер контролю часу увімкнення контактора
   END_VAR
BEGIN
   // =========================================================================================
   // ЛОГІКА КЕРУВАННЯ ЛІНІЙНИМ КОНТАКТОРОМ (ЛК) З РОЗДІЛЕННЯМ УМОВ СТАРТУ ТА РОБОТИ
   // =========================================================================================

   //------------------------------------------------------------------------------------------
   // 1. ЗБІР ПОСТІЙНО ДІЮЧИХ ЗАХИСТІВ ТА БЛОКУВАНЬ
   //------------------------------------------------------------------------------------------
   #qx_6HL2_SignalVoltage := #ix_6SF1_Breaker_6KV AND NOT #ix_6KV_VoltageCtrl_380V; // Вхідна напруга не в нормі

   // Базові апаратні умови готовності електрообладнання
   #stat_LC_Active := #ix_6SF1_Breaker_6KV
   AND #ix_6KV_VoltageCtrl_380V
   AND #ix_6SF5_HeaterBreaker
   AND #ix_6QF2_BrakeCircuitProt
   AND #ix_6QF3_TransfBreaker_6T1
   AND #ix_6QF4_TransfSecBreaker
   AND #ix_6SF2_CtrlCircuit_220V
   AND #ix_6SF4_OVP_Power_220V
   AND #ix_1QF1_BrakeRectifier_1YB1
   AND #ix_1QF2_BrakeRectifier_1YB2
   AND #ix_4QF1_BrakeCircuitProt
   AND #ix_9QF4_CabinetAux_220V;

   // Перевірка дозволів роботи механізмів (ручні приводи відключені / РП роз'єднані)
   #stat_LC_Active := #stat_LC_Active
   AND #is_Manual_interlock.LM_WP_disconn_brake
   AND #is_Manual_interlock.LM_WP_disconn_drive
   AND #is_Manual_interlock.TM_WP_disconn_drive
   AND #is_Manual_interlock.CM_WP_disconn_drive_1
   AND #is_Manual_interlock.CM_WP_disconn_drive_2;

   // Контроль кінцевих вимикачів руху крайніх положень
   #stat_LC_Active := #stat_LC_Active
   AND #is_MovePerm.Upward
   AND #is_MovePerm.Downward
   AND #is_MovePerm.Forward
   AND #is_MovePerm.Backward
   AND #is_MovePerm.Left
   AND #is_MovePerm.Right
   AND (#is_MovePerm.No_Pillar OR #is_SpeedPerm.Speed_normal_Bwd);

   // Інтеграція умов щодо сейсміки, мережі Profinet та пожежна тривога
   #stat_LC_Active := #stat_LC_Active
   AND NOT #ix_K3_SeismicAlarm
   AND #ix_Profinet_OK
   AND NOT #ix_FireAlarm;

   //------------------------------------------------------------------------------------------
   // 2. ЗАХИСТ ВІД НЕСАНКЦІОНОВАНОГО ПУСКУ (Нульовий захист)
   //------------------------------------------------------------------------------------------
   // Всі органи керування повинні бути відпущені для зняття стартового блокування
   IF NOT #ix_6K3_CmdStart
       AND NOT #is_RemCtrl.Btn_Up AND NOT #is_RemCtrl.Btn_Down
       AND NOT #is_RemCtrl.Btn_Fwd AND NOT #is_RemCtrl.Btn_Bwd
       AND NOT #is_RemCtrl.Btn_Left AND NOT #is_RemCtrl.Btn_Right
       AND #ix_6KV_VoltageCtrl_380V
       AND #ix_6SF5_HeaterBreaker
       AND #ix_6QF2_BrakeCircuitProt
       AND #ix_6QF3_TransfBreaker_6T1
       AND #ix_6QF4_TransfSecBreaker
       AND #ix_6SF2_CtrlCircuit_220V
       AND #ix_6SF4_OVP_Power_220V
       AND #ix_1QF1_BrakeRectifier_1YB1
       AND #ix_1QF2_BrakeRectifier_1YB2
       AND #ix_4QF1_BrakeCircuitProt
       AND #ix_9QF4_CabinetAux_220V
       AND #is_Manual_interlock.LM_WP_disconn_brake
       AND #is_Manual_interlock.LM_WP_disconn_drive
       AND #is_Manual_interlock.TM_WP_disconn_drive
       AND #is_Manual_interlock.CM_WP_disconn_drive_1
       AND #is_Manual_interlock.CM_WP_disconn_drive_2
       AND #is_MovePerm.Upward
       AND #is_MovePerm.Downward
       AND #is_MovePerm.Forward
       AND #is_MovePerm.Backward
       AND #is_MovePerm.Left
       AND #is_MovePerm.Right
       AND(#is_MovePerm.No_Pillar OR #is_SpeedPerm.Speed_normal_Bwd)
       AND NOT #ix_K3_SeismicAlarm
       AND #ix_Profinet_OK
       AND NOT #ix_FireAlarm
       AND NOT #qx_Alarm_Active
   THEN
       #stat_InterlockStartup := FALSE;
   END_IF;

   // Якщо сигнал 6К3 прийшов ДО виконання умов первинного прогріву чи готовності власних потреб — блокуємо включення
   IF #ix_6K3_CmdStart AND NOT #stat_InterlockStartup AND NOT #ix_6KM1_Feedback_LC THEN
       IF NOT #ix_9K2_CabinetHeating
           OR NOT #ix_9QF4_CabinetAux_220V
           OR #is_RemCtrl.Btn_Up OR #is_RemCtrl.Btn_Down
           OR #is_RemCtrl.Btn_Fwd OR #is_RemCtrl.Btn_Bwd
           OR #is_RemCtrl.Btn_Left OR #is_RemCtrl.Btn_Right
           OR NOT #ix_6KV_VoltageCtrl_380V
           OR NOT #ix_6SF5_HeaterBreaker
           OR NOT #ix_6QF2_BrakeCircuitProt
           OR NOT #ix_6QF3_TransfBreaker_6T1
           OR NOT #ix_6QF4_TransfSecBreaker
           OR NOT #ix_6SF2_CtrlCircuit_220V
           OR NOT #ix_6SF4_OVP_Power_220V
           OR NOT #ix_1QF1_BrakeRectifier_1YB1
           OR NOT #ix_1QF2_BrakeRectifier_1YB2
           OR NOT #ix_4QF1_BrakeCircuitProt
           OR NOT #is_Manual_interlock.LM_WP_disconn_brake
           OR NOT #is_Manual_interlock.LM_WP_disconn_drive
           OR NOT #is_Manual_interlock.TM_WP_disconn_drive
           OR NOT #is_Manual_interlock.CM_WP_disconn_drive_1
           OR NOT #is_Manual_interlock.CM_WP_disconn_drive_2
           OR NOT #is_MovePerm.Upward
           OR NOT #is_MovePerm.Downward
           OR NOT #is_MovePerm.Forward
           OR NOT #is_MovePerm.Backward
           OR NOT #is_MovePerm.Left
           OR NOT #is_MovePerm.Right
           OR NOT (#is_MovePerm.No_Pillar OR #is_SpeedPerm.Speed_normal_Bwd)
           OR #ix_K3_SeismicAlarm
           OR NOT #ix_Profinet_OK
           OR #ix_FireAlarm
           OR #qx_Alarm_Active
       THEN
           #stat_InterlockStartup := TRUE;
       END_IF;
   END_IF;

   // Передаємо стан внутрішнього прапора блокування на фізичний вихідний тег для HMI/ЛМИ
   #qx_Zero_Protection_Active := #stat_InterlockStartup;
   //------------------------------------------------------------------------------------------
   // 3. ФОРМУВАННЯ СИГНАЛІВ КЕРУВАННЯ 6K1 ТА 6K2 (З УРАХУВАННЯМ ДИНАМІЧНИХ УМОВ)
   //------------------------------------------------------------------------------------------
   // Перевірка умов утримання ланцюга 6K2:
   // Для включення/утримання потрібні: команда 6К3, базові захисти, відсутність аварій + виконання динамічної умови:
   // (Контактор уже сидить OR (Шафа прогріта AND Автомат власних потреб включений))
   IF #ix_6K3_CmdStart
       AND #stat_LC_Active
       AND NOT #stat_InterlockStartup
       AND (#stat_AlarmReg = 16#0000)
       AND (#ix_6KM1_Feedback_LC OR #ix_9K2_CabinetHeating) THEN

       #qx_6K2_Hold_LC := TRUE; // 6K2: Постійний сигнал утримання активний

       // 6K1 (Дозвіл включення): Видається тільки якщо контактор ще фізично НЕ замкнувся
       IF NOT #ix_6KM1_Feedback_LC THEN
           #qx_6K1_Permit_LC := TRUE;
       ELSE
           #qx_6K1_Permit_LC := FALSE; // Шунування: після отримання зворотного зв'язку знімаємо 6K1
       END_IF;
   ELSE
       // Беззумовне відключення обох каналів при знятті 6К3 або аварії
       #qx_6K2_Hold_LC := FALSE;
       #qx_6K1_Permit_LC := FALSE;
   END_IF;

   #qx_6HL1_SignalStart := #ix_6KM1_Feedback_LC;

   //------------------------------------------------------------------------------------------
   // 4. КОНТРОЛЬ ЗАХИСТІВ ТА ДІАГНОСТИКА АВАРІЙНИХ ПОДІЙ
   //------------------------------------------------------------------------------------------
   // Таймер контролю замикання аналізує вихід 6K1
   #stat_TimerFeedback(IN := #qx_6K2_Hold_LC AND NOT #ix_6KM1_Feedback_LC,
                       PT := T#2s);

   IF #stat_TimerFeedback.Q THEN
       #stat_AlarmReg.%X0 := TRUE; // Подія 0: Таймаут увімкнення контактора 6KM1
   END_IF;

   // Контроль контактора кіл керування 220В (6KM2)
   #stat_TimerFeedback_Con(IN:=#ix_6KM1_Feedback_LC AND NOT #ix_6KM2_Feedback_Ctrl220,
                           PT:=T#2s);

   IF #stat_TimerFeedback_Con.Q THEN
       #stat_AlarmReg.%X1 := TRUE; // Подія 1: Відсутність або зникнення сигналу 6КМ2
   END_IF;

   // Контроль логічної колізії (зворотний зв'язок є, а команди утримання ПЛК немає)
   #stat_TimerFeedback_LC(IN:=NOT #qx_6K2_Hold_LC AND #ix_6KM1_Feedback_LC,
                          PT:=T#2s);

   IF #stat_TimerFeedback_LC.Q THEN
       #stat_AlarmReg.%X2 := TRUE; // Подія 2: Спонтанне замикання контактора без команди
   END_IF;

   // Зовнішнє аварійне відключення під час роботи
   IF NOT #stat_LC_Active AND #ix_6KM1_Feedback_LC THEN
       #stat_AlarmReg.%X3 := TRUE; // Подія 3: Спрацювання постійних захистів/кінцевиків під час роботи
   END_IF;

   //------------------------------------------------------------------------------------------
   // 5. ПОБІТОВА ФІКСАЦІЯ ВСІХ ПОДІЙ У СЛОВА QW_TRIP_1 ТА QW_TRIP_2 ПРИ ВІДКЛЮЧЕННІ
   //------------------------------------------------------------------------------------------
   //
   #qw_Trip_1.%X0 := #stat_AlarmReg.%X0;          // Подія 0: Таймаут увімкнення контактора 6KM1
   #qw_Trip_1.%X1 := #stat_AlarmReg.%X1;          // Подія 1: Відсутній або зник сигнал контактора 6КМ2
   IF #stat_Prev_KM1_Feedback AND NOT #ix_6KM1_Feedback_LC THEN

       #qw_Trip_1 := 16#0000;
       #qw_Trip_2 := 16#0000;

       // --- ЗАПОВНЕННЯ СЛОВА QW_TRIP_1 (Події 2..15) ---

       #qw_Trip_1.%X2 := NOT #ix_6SF1_Breaker_6KV;       // Подія 2: Вимкнено вимикач живлення 6KV
       #qw_Trip_1.%X3 := NOT #ix_6KV_VoltageCtrl_380V;   // Подія 3: Вхідна напруга не в нормі
       #qw_Trip_1.%X4 := NOT #ix_6SF5_HeaterBreaker;     // Подія 4: Вимкнено автомат обігріву шафи
       #qw_Trip_1.%X5 := NOT #ix_6QF2_BrakeCircuitProt;  // Подія 5: Вимкнено автомат захисту кіл гальм
       #qw_Trip_1.%X6 := NOT #ix_6QF3_TransfBreaker_6T1; // Подія 6: Вимкнено вимикач трансформатора 6T1
       #qw_Trip_1.%X7 := NOT #ix_6QF4_TransfSecBreaker;  // Подія 7: Вимкнено автомат вторинних кіл 6T1
       #qw_Trip_1.%X8 := NOT #ix_6SF2_CtrlCircuit_220V;  // Подія 8: Вимкнено вимикач кіл управління 220В
       #qw_Trip_1.%X9 := NOT #ix_6SF4_OVP_Power_220V;    // Подія 9: Вимкнено автомат живлення ОВП 220В
       #qw_Trip_1.%X10 := NOT #ix_9QF4_CabinetAux_220V;   // Подія 10: Відсутність готовності власних потреб шафи 220В
       #qw_Trip_1.%X11 := NOT #ix_1QF1_BrakeRectifier_1YB1;// Подія 11: Аварія захисту випрямляча гальма 1YB1
       #qw_Trip_1.%X12 := NOT #ix_1QF2_BrakeRectifier_1YB2;// Подія 12: Аварія захисту випрямляча гальма 1YB2
       #qw_Trip_1.%X13 := NOT #ix_4QF1_BrakeCircuitProt; // Подія 13: Аварія захисту кіл гальм механізму 4
       #qw_Trip_1.%X14 := NOT #is_Manual_interlock.LM_WP_disconn_brake;    // Подія 14: Відсутній дозвіл від гальма 1YB2
       #qw_Trip_1.%X15 := NOT #is_Manual_interlock.LM_WP_disconn_drive;   // Подія 15: Ручний привід підйому не відключено

       // --- ЗАПОВНЕННЯ СЛОВА QW_TRIP_2 (Події 16..31) ---
       #qw_Trip_2.%X0 := NOT #is_Manual_interlock.TM_WP_disconn_drive; // Подія 16: Ручний привід візка не роз'єднано
       #qw_Trip_2.%X1 := NOT #is_Manual_interlock.CM_WP_disconn_drive_1; // Подія 17: Ручний привід моста 1 не роз'єднано
       #qw_Trip_2.%X2 := NOT #is_Manual_interlock.CM_WP_disconn_drive_2; // Подія 18: Ручний привід моста 2 не роз'єднано
       #qw_Trip_2.%X3 := NOT #is_MovePerm.Upward;       // Подія 19: Спрацював кінцевик Підйом ВГОРУ
       #qw_Trip_2.%X4 := NOT #is_MovePerm.Downward;     // Подія 20: Спрацював кінцевик Підйом ВНИЗ
       #qw_Trip_2.%X5 := NOT #is_MovePerm.Forward;  // Подія 21: Спрацював кінцевик Візок ВПЕРЕД
       #qw_Trip_2.%X6 := NOT #is_MovePerm.Backward; // Подія 22: Спрацював кінцевик Візок НАЗАД
       #qw_Trip_2.%X7 := NOT #is_MovePerm.Left;      // Подія 23: Спрацював кінцевик Мост ВЛІВО
       #qw_Trip_2.%X8 := NOT #is_MovePerm.Right;     // Подія 24: Спрацював кінцевик Мост ВПРАВО
       #qw_Trip_2.%X9 := #ix_K3_SeismicAlarm;           // Подія 25: Спрацював сигнал сейсмодатчика 9К3
       #qw_Trip_2.%X10 := NOT #ix_Profinet_OK;           // Подія 26: Критична помилка мережі Profinet
       #qw_Trip_2.%X11 := NOT (#is_MovePerm.No_Pillar OR #is_SpeedPerm.Speed_normal_Bwd); //Подія 27:Візок у зоні колони
       #qw_Trip_2.%X12 := #ix_FireAlarm; //Подія 28: Пожежна тривога
   END_IF;

   #stat_Prev_KM1_Feedback := #ix_6KM1_Feedback_LC;

   //------------------------------------------------------------------------------------------
   // 6. КВІТУВАННЯ ТА СКИДАННЯ ПОМИЛОК
   //------------------------------------------------------------------------------------------
   IF #ix_Ack THEN
       #stat_AlarmReg := 16#0000;


       #qw_Trip_1 := 16#0000;
       #qw_Trip_2 := 16#0000;
   END_IF;

   #qx_Alarm_Active := (#stat_AlarmReg <> 16#0000);
   #qw_Alarm_Code := #stat_AlarmReg;
END_FUNCTION_BLOCK

FUNCTION_BLOCK "FB_PSM_Messages"   // FB21, LAD
{ S7_Optimized_Access := 'TRUE' }
VERSION : 0.1
   VAR
      ssfbTon1 : IEC_TIMER;
      ssfbTon2 : IEC_TIMER;
      sxMode : Bool;   // Операційний біт (0 - онлайн, 1 - офлайн)
      sxStartUp : Bool;   // Стартап біт (0 - при старті, 1 - під час роботи)
      sxLifeBit : Bool;   // Лайфбіт
      ssfbHMI_w1 : "FB_DigIn_16_XOR";
      ssfbHMI_w2 : "FB_DigIn_16_XOR";
      ssfbHMI_w3 : "FB_DigIn_16_XOR";
      ssfbHMI_w4 : "FB_DigIn_16_XOR";
      ssfbHMI_w5 : "FB_DigIn_16_XOR";
      ssfbHMI_w6 : "FB_DigIn_16_XOR";
   END_VAR
   VAR_TEMP
      txProfinetOk : Bool;   // Зв'язок по мережі профінет
      txNullBlockOk : Bool;   // Нульове блокування присутнє
   END_VAR
BEGIN

REGION Network 1: Операційний біт (0 - онлайн, 1 - офлайн)
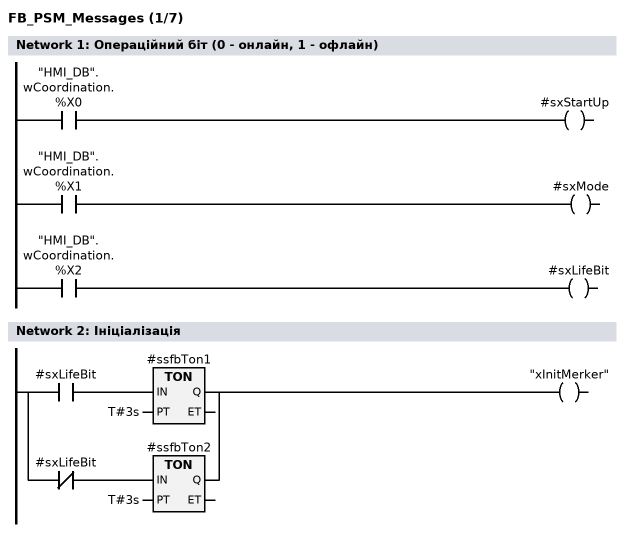
   RUNG wire#powerrail
      Contact( "HMI_DB".wCoordination.%X0 )
      Coil( #sxStartUp )
   END_RUNG
   RUNG wire#powerrail
      Contact( "HMI_DB".wCoordination.%X1 )
      Coil( #sxMode )
   END_RUNG
   RUNG wire#powerrail
      Contact( "HMI_DB".wCoordination.%X2 )
      Coil( #sxLifeBit )
   END_RUNG
   // the same network as SCL:
   #sxStartUp := "HMI_DB".wCoordination.%X0;
   #sxMode := "HMI_DB".wCoordination.%X1;
   #sxLifeBit := "HMI_DB".wCoordination.%X2;
END_REGION

REGION Network 2: Ініціалізація
   #ssfbTon1.TON(IN := #sxLifeBit, PT := T#3s);
   #ssfbTon2.TON(IN := NOT #sxLifeBit, PT := T#3s);
   "xInitMerker" := #ssfbTon1.Q OR #ssfbTon2.Q;
END_REGION

REGION Network 3: Перше слово повідомлень
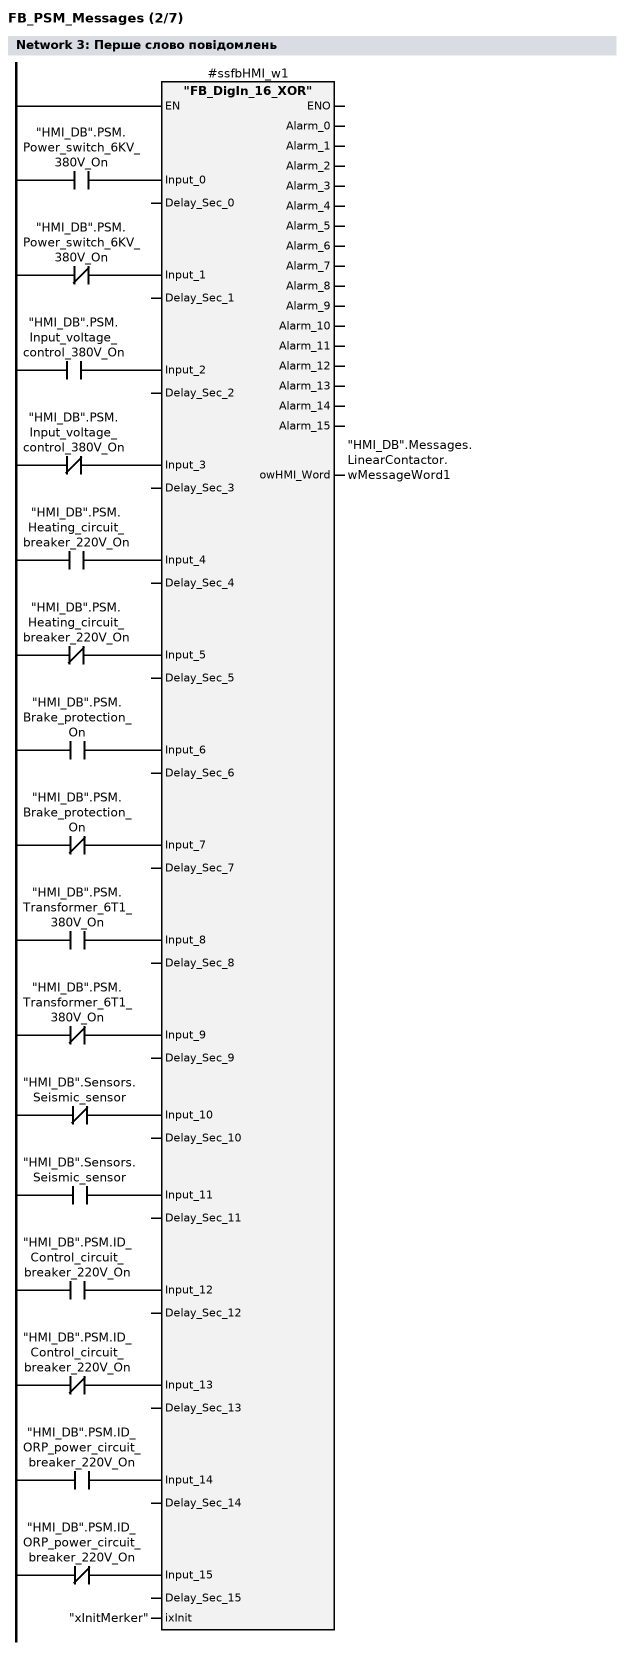
   RUNG wire#powerrail
      #ssfbHMI_w1(Input_0 := wire#w1, Input_1 := wire#w2, Input_2 := wire#w3, Input_3 := wire#w4, Input_4 := wire#w5, Input_5 := wire#w6, Input_6 := wire#w7, Input_7 := wire#w8, Input_8 := wire#w9, Input_9 := wire#w10, Input_10 := wire#w11, Input_11 := wire#w12, Input_12 := wire#w13, Input_13 := wire#w14, Input_14 := wire#w15, Input_15 := wire#w16, Delay_Sec_0 :=, Delay_Sec_1 :=, Delay_Sec_2 :=, Delay_Sec_3 :=, Delay_Sec_4 :=, Delay_Sec_5 :=, Delay_Sec_6 :=, Delay_Sec_7 :=, Delay_Sec_8 :=, Delay_Sec_9 :=, Delay_Sec_10 :=, Delay_Sec_11 :=, Delay_Sec_12 :=, Delay_Sec_13 :=, Delay_Sec_14 :=, Delay_Sec_15 :=, ixInit := "xInitMerker", Alarm_0 =>, Alarm_1 =>, Alarm_2 =>, Alarm_3 =>, Alarm_4 =>, Alarm_5 =>, Alarm_6 =>, Alarm_7 =>, Alarm_8 =>, Alarm_9 =>, Alarm_10 =>, Alarm_11 =>, Alarm_12 =>, Alarm_13 =>, Alarm_14 =>, Alarm_15 =>, owHMI_Word => "HMI_DB".Messages.LinearContactor.wMessageWord1)
   END_RUNG
   RUNG wire#powerrail
      Contact( "HMI_DB".PSM.Power_switch_6KV_380V_On )
   END_RUNG wire#w1
   RUNG wire#powerrail
      I_Contact( "HMI_DB".PSM.Power_switch_6KV_380V_On )
   END_RUNG wire#w2
   RUNG wire#powerrail
      Contact( "HMI_DB".PSM.Input_voltage_control_380V_On )
   END_RUNG wire#w3
   RUNG wire#powerrail
      I_Contact( "HMI_DB".PSM.Input_voltage_control_380V_On )
   END_RUNG wire#w4
   RUNG wire#powerrail
      Contact( "HMI_DB".PSM.Heating_circuit_breaker_220V_On )
   END_RUNG wire#w5
   RUNG wire#powerrail
      I_Contact( "HMI_DB".PSM.Heating_circuit_breaker_220V_On )
   END_RUNG wire#w6
   RUNG wire#powerrail
      Contact( "HMI_DB".PSM.Brake_protection_On )
   END_RUNG wire#w7
   RUNG wire#powerrail
      I_Contact( "HMI_DB".PSM.Brake_protection_On )
   END_RUNG wire#w8
   RUNG wire#powerrail
      Contact( "HMI_DB".PSM.Transformer_6T1_380V_On )
   END_RUNG wire#w9
   RUNG wire#powerrail
      I_Contact( "HMI_DB".PSM.Transformer_6T1_380V_On )
   END_RUNG wire#w10
   RUNG wire#powerrail
      I_Contact( "HMI_DB".Sensors.Seismic_sensor )
   END_RUNG wire#w11
   RUNG wire#powerrail
      Contact( "HMI_DB".Sensors.Seismic_sensor )
   END_RUNG wire#w12
   RUNG wire#powerrail
      Contact( "HMI_DB".PSM.ID_Control_circuit_breaker_220V_On )
   END_RUNG wire#w13
   RUNG wire#powerrail
      I_Contact( "HMI_DB".PSM.ID_Control_circuit_breaker_220V_On )
   END_RUNG wire#w14
   RUNG wire#powerrail
      Contact( "HMI_DB".PSM.ID_ORP_power_circuit_breaker_220V_On )
   END_RUNG wire#w15
   RUNG wire#powerrail
      I_Contact( "HMI_DB".PSM.ID_ORP_power_circuit_breaker_220V_On )
   END_RUNG wire#w16
   // the same network as SCL:
   #ssfbHMI_w1(Input_0 := "HMI_DB".PSM.Power_switch_6KV_380V_On,   // "FB_DigIn_16_XOR"
               Input_1 := NOT "HMI_DB".PSM.Power_switch_6KV_380V_On,
               Input_2 := "HMI_DB".PSM.Input_voltage_control_380V_On,
               Input_3 := NOT "HMI_DB".PSM.Input_voltage_control_380V_On,
               Input_4 := "HMI_DB".PSM.Heating_circuit_breaker_220V_On,
               Input_5 := NOT "HMI_DB".PSM.Heating_circuit_breaker_220V_On,
               Input_6 := "HMI_DB".PSM.Brake_protection_On,
               Input_7 := NOT "HMI_DB".PSM.Brake_protection_On,
               Input_8 := "HMI_DB".PSM.Transformer_6T1_380V_On,
               Input_9 := NOT "HMI_DB".PSM.Transformer_6T1_380V_On,
               Input_10 := NOT "HMI_DB".Sensors.Seismic_sensor,
               Input_11 := "HMI_DB".Sensors.Seismic_sensor,
               Input_12 := "HMI_DB".PSM.ID_Control_circuit_breaker_220V_On,
               Input_13 := NOT "HMI_DB".PSM.ID_Control_circuit_breaker_220V_On,
               Input_14 := "HMI_DB".PSM.ID_ORP_power_circuit_breaker_220V_On,
               Input_15 := NOT "HMI_DB".PSM.ID_ORP_power_circuit_breaker_220V_On,
               ixInit := "xInitMerker",
               owHMI_Word => "HMI_DB".Messages.LinearContactor.wMessageWord1);
END_REGION

REGION Network 4: Друге слово повідомлень
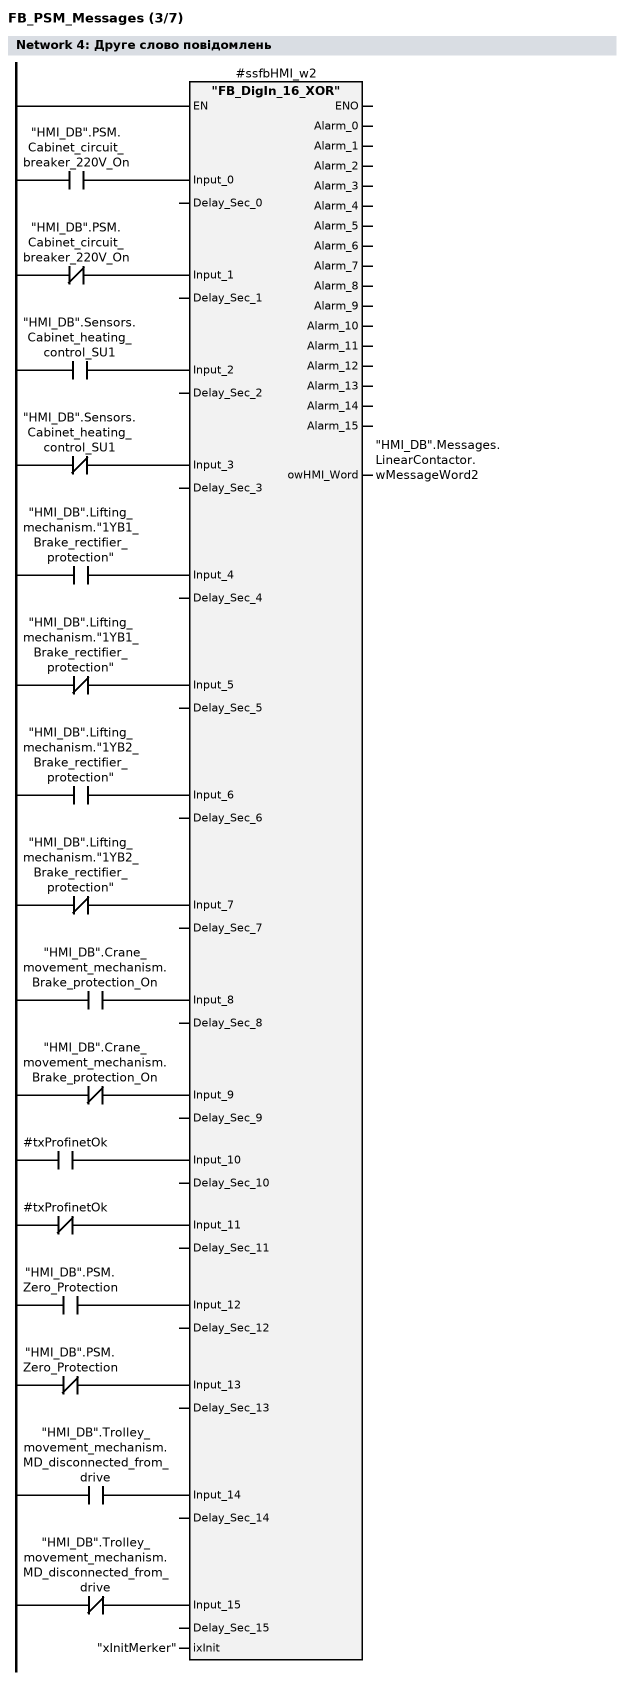
   RUNG wire#powerrail
      #ssfbHMI_w2(Input_0 := wire#w1, Input_1 := wire#w2, Input_2 := wire#w3, Input_3 := wire#w4, Input_4 := wire#w5, Input_5 := wire#w6, Input_6 := wire#w7, Input_7 := wire#w8, Input_8 := wire#w9, Input_9 := wire#w10, Input_10 := wire#w11, Input_11 := wire#w12, Input_12 := wire#w13, Input_13 := wire#w14, Input_14 := wire#w15, Input_15 := wire#w16, Delay_Sec_0 :=, Delay_Sec_1 :=, Delay_Sec_2 :=, Delay_Sec_3 :=, Delay_Sec_4 :=, Delay_Sec_5 :=, Delay_Sec_6 :=, Delay_Sec_7 :=, Delay_Sec_8 :=, Delay_Sec_9 :=, Delay_Sec_10 :=, Delay_Sec_11 :=, Delay_Sec_12 :=, Delay_Sec_13 :=, Delay_Sec_14 :=, Delay_Sec_15 :=, ixInit := "xInitMerker", Alarm_0 =>, Alarm_1 =>, Alarm_2 =>, Alarm_3 =>, Alarm_4 =>, Alarm_5 =>, Alarm_6 =>, Alarm_7 =>, Alarm_8 =>, Alarm_9 =>, Alarm_10 =>, Alarm_11 =>, Alarm_12 =>, Alarm_13 =>, Alarm_14 =>, Alarm_15 =>, owHMI_Word => "HMI_DB".Messages.LinearContactor.wMessageWord2)
   END_RUNG
   RUNG wire#powerrail
      Contact( "HMI_DB".PSM.Cabinet_circuit_breaker_220V_On )
   END_RUNG wire#w1
   RUNG wire#powerrail
      I_Contact( "HMI_DB".PSM.Cabinet_circuit_breaker_220V_On )
   END_RUNG wire#w2
   RUNG wire#powerrail
      Contact( "HMI_DB".Sensors.Cabinet_heating_control_SU1 )
   END_RUNG wire#w3
   RUNG wire#powerrail
      I_Contact( "HMI_DB".Sensors.Cabinet_heating_control_SU1 )
   END_RUNG wire#w4
   RUNG wire#powerrail
      Contact( "HMI_DB".Lifting_mechanism."1YB1_Brake_rectifier_protection" )
   END_RUNG wire#w5
   RUNG wire#powerrail
      I_Contact( "HMI_DB".Lifting_mechanism."1YB1_Brake_rectifier_protection" )
   END_RUNG wire#w6
   RUNG wire#powerrail
      Contact( "HMI_DB".Lifting_mechanism."1YB2_Brake_rectifier_protection" )
   END_RUNG wire#w7
   RUNG wire#powerrail
      I_Contact( "HMI_DB".Lifting_mechanism."1YB2_Brake_rectifier_protection" )
   END_RUNG wire#w8
   RUNG wire#powerrail
      Contact( "HMI_DB".Crane_movement_mechanism.Brake_protection_On )
   END_RUNG wire#w9
   RUNG wire#powerrail
      I_Contact( "HMI_DB".Crane_movement_mechanism.Brake_protection_On )
   END_RUNG wire#w10
   RUNG wire#powerrail
      Contact( #txProfinetOk )
   END_RUNG wire#w11
   RUNG wire#powerrail
      I_Contact( #txProfinetOk )
   END_RUNG wire#w12
   RUNG wire#powerrail
      Contact( "HMI_DB".PSM.Zero_Protection )
   END_RUNG wire#w13
   RUNG wire#powerrail
      I_Contact( "HMI_DB".PSM.Zero_Protection )
   END_RUNG wire#w14
   RUNG wire#powerrail
      Contact( "HMI_DB".Trolley_movement_mechanism.MD_disconnected_from_drive )
   END_RUNG wire#w15
   RUNG wire#powerrail
      I_Contact( "HMI_DB".Trolley_movement_mechanism.MD_disconnected_from_drive )
   END_RUNG wire#w16
   // the same network as SCL:
   #ssfbHMI_w2(Input_0 := "HMI_DB".PSM.Cabinet_circuit_breaker_220V_On,   // "FB_DigIn_16_XOR"
               Input_1 := NOT "HMI_DB".PSM.Cabinet_circuit_breaker_220V_On,
               Input_2 := "HMI_DB".Sensors.Cabinet_heating_control_SU1,
               Input_3 := NOT "HMI_DB".Sensors.Cabinet_heating_control_SU1,
               Input_4 := "HMI_DB".Lifting_mechanism."1YB1_Brake_rectifier_protection",
               Input_5 := NOT "HMI_DB".Lifting_mechanism."1YB1_Brake_rectifier_protection",
               Input_6 := "HMI_DB".Lifting_mechanism."1YB2_Brake_rectifier_protection",
               Input_7 := NOT "HMI_DB".Lifting_mechanism."1YB2_Brake_rectifier_protection",
               Input_8 := "HMI_DB".Crane_movement_mechanism.Brake_protection_On,
               Input_9 := NOT "HMI_DB".Crane_movement_mechanism.Brake_protection_On,
               Input_10 := #txProfinetOk,
               Input_11 := NOT #txProfinetOk,
               Input_12 := "HMI_DB".PSM.Zero_Protection,
               Input_13 := NOT "HMI_DB".PSM.Zero_Protection,
               Input_14 := "HMI_DB".Trolley_movement_mechanism.MD_disconnected_from_drive,
               Input_15 := NOT "HMI_DB".Trolley_movement_mechanism.MD_disconnected_from_drive,
               ixInit := "xInitMerker",
               owHMI_Word => "HMI_DB".Messages.LinearContactor.wMessageWord2);
END_REGION

REGION Network 5: Третє слово повідомлень
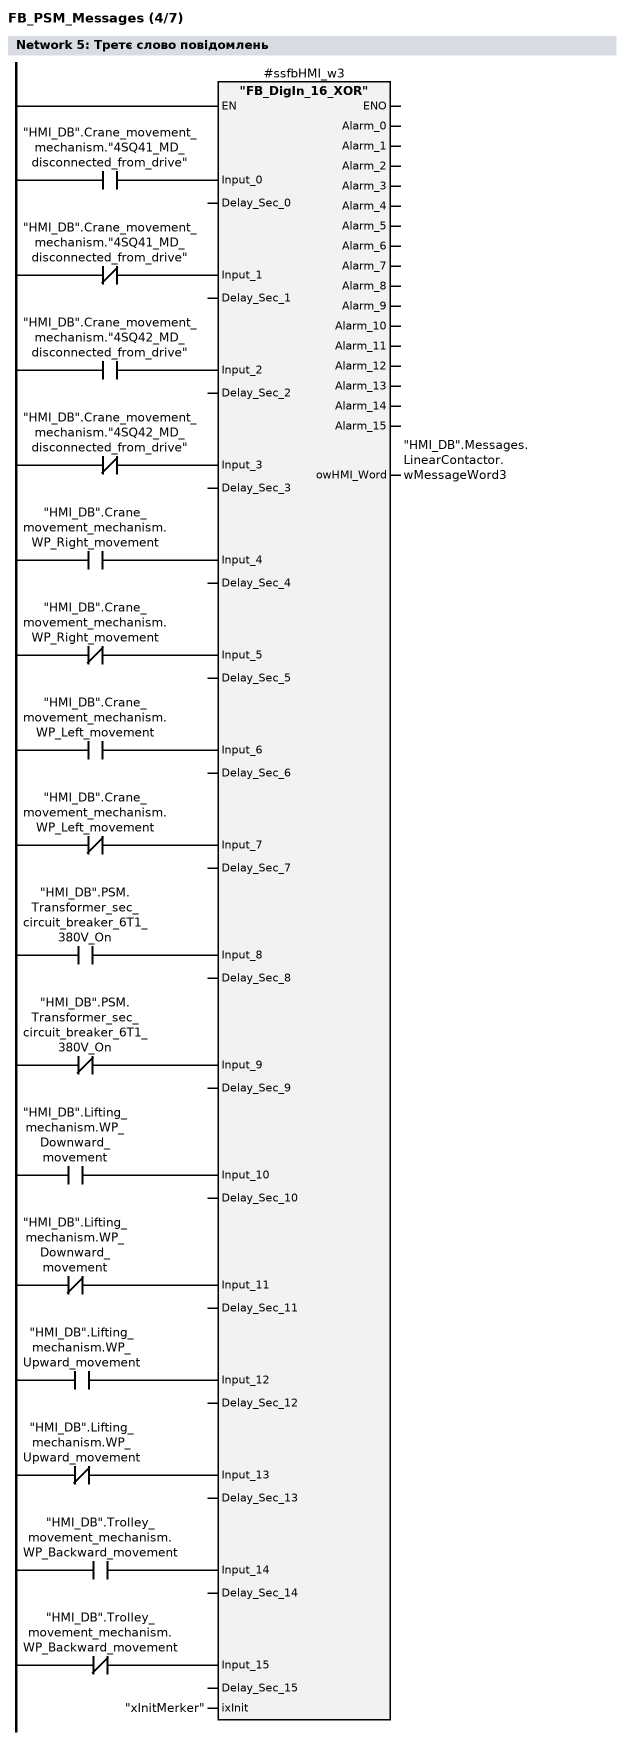
   RUNG wire#powerrail
      #ssfbHMI_w3(Input_0 := wire#w1, Input_1 := wire#w2, Input_2 := wire#w3, Input_3 := wire#w4, Input_4 := wire#w5, Input_5 := wire#w6, Input_6 := wire#w7, Input_7 := wire#w8, Input_8 := wire#w9, Input_9 := wire#w10, Input_10 := wire#w11, Input_11 := wire#w12, Input_12 := wire#w13, Input_13 := wire#w14, Input_14 := wire#w15, Input_15 := wire#w16, Delay_Sec_0 :=, Delay_Sec_1 :=, Delay_Sec_2 :=, Delay_Sec_3 :=, Delay_Sec_4 :=, Delay_Sec_5 :=, Delay_Sec_6 :=, Delay_Sec_7 :=, Delay_Sec_8 :=, Delay_Sec_9 :=, Delay_Sec_10 :=, Delay_Sec_11 :=, Delay_Sec_12 :=, Delay_Sec_13 :=, Delay_Sec_14 :=, Delay_Sec_15 :=, ixInit := "xInitMerker", Alarm_0 =>, Alarm_1 =>, Alarm_2 =>, Alarm_3 =>, Alarm_4 =>, Alarm_5 =>, Alarm_6 =>, Alarm_7 =>, Alarm_8 =>, Alarm_9 =>, Alarm_10 =>, Alarm_11 =>, Alarm_12 =>, Alarm_13 =>, Alarm_14 =>, Alarm_15 =>, owHMI_Word => "HMI_DB".Messages.LinearContactor.wMessageWord3)
   END_RUNG
   RUNG wire#powerrail
      Contact( "HMI_DB".Crane_movement_mechanism."4SQ41_MD_disconnected_from_drive" )
   END_RUNG wire#w1
   RUNG wire#powerrail
      I_Contact( "HMI_DB".Crane_movement_mechanism."4SQ41_MD_disconnected_from_drive" )
   END_RUNG wire#w2
   RUNG wire#powerrail
      Contact( "HMI_DB".Crane_movement_mechanism."4SQ42_MD_disconnected_from_drive" )
   END_RUNG wire#w3
   RUNG wire#powerrail
      I_Contact( "HMI_DB".Crane_movement_mechanism."4SQ42_MD_disconnected_from_drive" )
   END_RUNG wire#w4
   RUNG wire#powerrail
      Contact( "HMI_DB".Crane_movement_mechanism.WP_Right_movement )
   END_RUNG wire#w5
   RUNG wire#powerrail
      I_Contact( "HMI_DB".Crane_movement_mechanism.WP_Right_movement )
   END_RUNG wire#w6
   RUNG wire#powerrail
      Contact( "HMI_DB".Crane_movement_mechanism.WP_Left_movement )
   END_RUNG wire#w7
   RUNG wire#powerrail
      I_Contact( "HMI_DB".Crane_movement_mechanism.WP_Left_movement )
   END_RUNG wire#w8
   RUNG wire#powerrail
      Contact( "HMI_DB".PSM.Transformer_sec_circuit_breaker_6T1_380V_On )
   END_RUNG wire#w9
   RUNG wire#powerrail
      I_Contact( "HMI_DB".PSM.Transformer_sec_circuit_breaker_6T1_380V_On )
   END_RUNG wire#w10
   RUNG wire#powerrail
      Contact( "HMI_DB".Lifting_mechanism.WP_Downward_movement )
   END_RUNG wire#w11
   RUNG wire#powerrail
      I_Contact( "HMI_DB".Lifting_mechanism.WP_Downward_movement )
   END_RUNG wire#w12
   RUNG wire#powerrail
      Contact( "HMI_DB".Lifting_mechanism.WP_Upward_movement )
   END_RUNG wire#w13
   RUNG wire#powerrail
      I_Contact( "HMI_DB".Lifting_mechanism.WP_Upward_movement )
   END_RUNG wire#w14
   RUNG wire#powerrail
      Contact( "HMI_DB".Trolley_movement_mechanism.WP_Backward_movement )
   END_RUNG wire#w15
   RUNG wire#powerrail
      I_Contact( "HMI_DB".Trolley_movement_mechanism.WP_Backward_movement )
   END_RUNG wire#w16
   // the same network as SCL:
   #ssfbHMI_w3(Input_0 := "HMI_DB".Crane_movement_mechanism."4SQ41_MD_disconnected_from_drive",   // "FB_DigIn_16_XOR"
               Input_1 := NOT "HMI_DB".Crane_movement_mechanism."4SQ41_MD_disconnected_from_drive",
               Input_2 := "HMI_DB".Crane_movement_mechanism."4SQ42_MD_disconnected_from_drive",
               Input_3 := NOT "HMI_DB".Crane_movement_mechanism."4SQ42_MD_disconnected_from_drive",
               Input_4 := "HMI_DB".Crane_movement_mechanism.WP_Right_movement,
               Input_5 := NOT "HMI_DB".Crane_movement_mechanism.WP_Right_movement,
               Input_6 := "HMI_DB".Crane_movement_mechanism.WP_Left_movement,
               Input_7 := NOT "HMI_DB".Crane_movement_mechanism.WP_Left_movement,
               Input_8 := "HMI_DB".PSM.Transformer_sec_circuit_breaker_6T1_380V_On,
               Input_9 := NOT "HMI_DB".PSM.Transformer_sec_circuit_breaker_6T1_380V_On,
               Input_10 := "HMI_DB".Lifting_mechanism.WP_Downward_movement,
               Input_11 := NOT "HMI_DB".Lifting_mechanism.WP_Downward_movement,
               Input_12 := "HMI_DB".Lifting_mechanism.WP_Upward_movement,
               Input_13 := NOT "HMI_DB".Lifting_mechanism.WP_Upward_movement,
               Input_14 := "HMI_DB".Trolley_movement_mechanism.WP_Backward_movement,
               Input_15 := NOT "HMI_DB".Trolley_movement_mechanism.WP_Backward_movement,
               ixInit := "xInitMerker",
               owHMI_Word => "HMI_DB".Messages.LinearContactor.wMessageWord3);
END_REGION

REGION Network 6: Четверте слово повідомлень
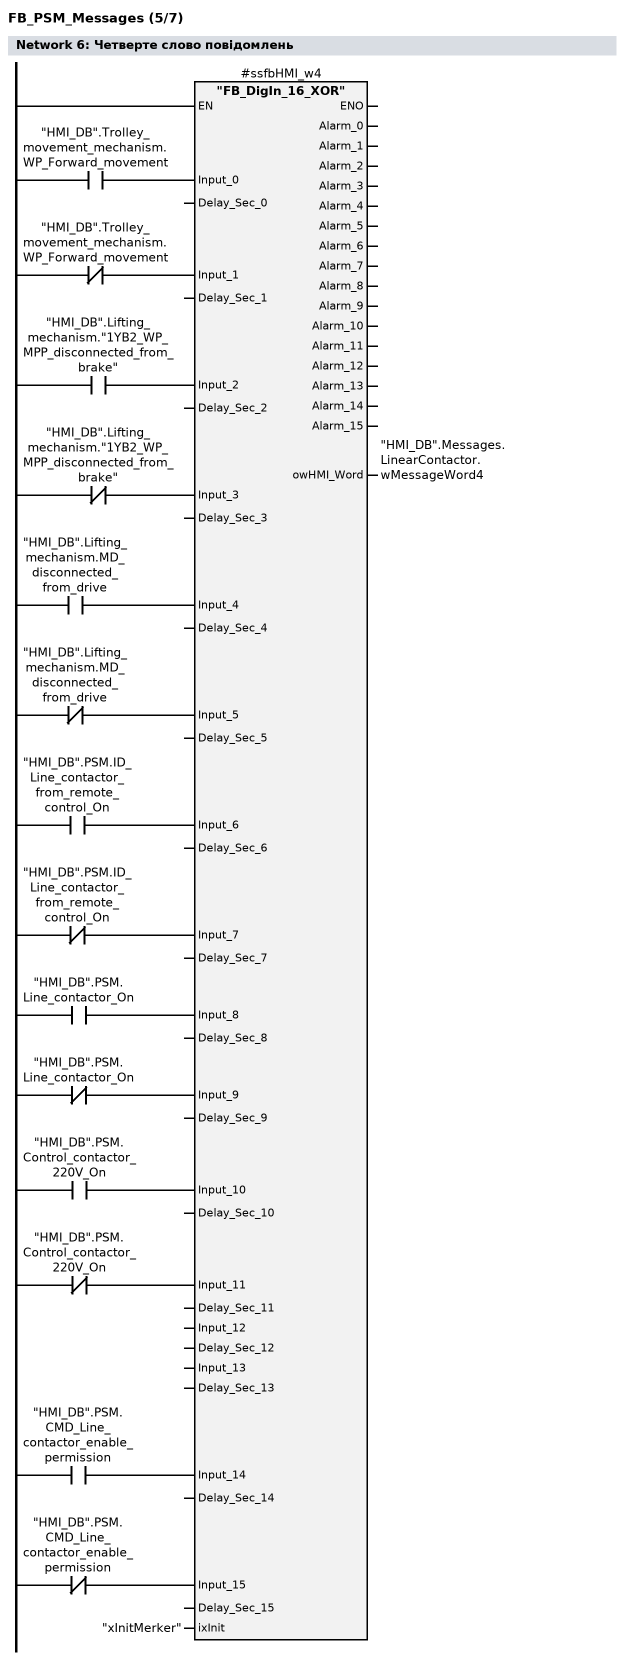
   RUNG wire#powerrail
      #ssfbHMI_w4(Input_0 := wire#w1, Input_1 := wire#w2, Input_2 := wire#w3, Input_3 := wire#w4, Input_4 := wire#w5, Input_5 := wire#w6, Input_6 := wire#w7, Input_7 := wire#w8, Input_8 := wire#w9, Input_9 := wire#w10, Input_10 := wire#w11, Input_11 := wire#w12, Input_14 := wire#w13, Input_15 := wire#w14, Delay_Sec_0 :=, Delay_Sec_1 :=, Delay_Sec_2 :=, Delay_Sec_3 :=, Delay_Sec_4 :=, Delay_Sec_5 :=, Delay_Sec_6 :=, Delay_Sec_7 :=, Delay_Sec_8 :=, Delay_Sec_9 :=, Delay_Sec_10 :=, Delay_Sec_11 :=, Input_12 :=, Delay_Sec_12 :=, Input_13 :=, Delay_Sec_13 :=, Delay_Sec_14 :=, Delay_Sec_15 :=, ixInit := "xInitMerker", Alarm_0 =>, Alarm_1 =>, Alarm_2 =>, Alarm_3 =>, Alarm_4 =>, Alarm_5 =>, Alarm_6 =>, Alarm_7 =>, Alarm_8 =>, Alarm_9 =>, Alarm_10 =>, Alarm_11 =>, Alarm_12 =>, Alarm_13 =>, Alarm_14 =>, Alarm_15 =>, owHMI_Word => "HMI_DB".Messages.LinearContactor.wMessageWord4)
   END_RUNG
   RUNG wire#powerrail
      Contact( "HMI_DB".Trolley_movement_mechanism.WP_Forward_movement )
   END_RUNG wire#w1
   RUNG wire#powerrail
      I_Contact( "HMI_DB".Trolley_movement_mechanism.WP_Forward_movement )
   END_RUNG wire#w2
   RUNG wire#powerrail
      Contact( "HMI_DB".Lifting_mechanism."1YB2_WP_MPP_disconnected_from_brake" )
   END_RUNG wire#w3
   RUNG wire#powerrail
      I_Contact( "HMI_DB".Lifting_mechanism."1YB2_WP_MPP_disconnected_from_brake" )
   END_RUNG wire#w4
   RUNG wire#powerrail
      Contact( "HMI_DB".Lifting_mechanism.MD_disconnected_from_drive )
   END_RUNG wire#w5
   RUNG wire#powerrail
      I_Contact( "HMI_DB".Lifting_mechanism.MD_disconnected_from_drive )
   END_RUNG wire#w6
   RUNG wire#powerrail
      Contact( "HMI_DB".PSM.ID_Line_contactor_from_remote_control_On )
   END_RUNG wire#w7
   RUNG wire#powerrail
      I_Contact( "HMI_DB".PSM.ID_Line_contactor_from_remote_control_On )
   END_RUNG wire#w8
   RUNG wire#powerrail
      Contact( "HMI_DB".PSM.Line_contactor_On )
   END_RUNG wire#w9
   RUNG wire#powerrail
      I_Contact( "HMI_DB".PSM.Line_contactor_On )
   END_RUNG wire#w10
   RUNG wire#powerrail
      Contact( "HMI_DB".PSM.Control_contactor_220V_On )
   END_RUNG wire#w11
   RUNG wire#powerrail
      I_Contact( "HMI_DB".PSM.Control_contactor_220V_On )
   END_RUNG wire#w12
   RUNG wire#powerrail
      Contact( "HMI_DB".PSM.CMD_Line_contactor_enable_permission )
   END_RUNG wire#w13
   RUNG wire#powerrail
      I_Contact( "HMI_DB".PSM.CMD_Line_contactor_enable_permission )
   END_RUNG wire#w14
   // the same network as SCL:
   #ssfbHMI_w4(Input_0 := "HMI_DB".Trolley_movement_mechanism.WP_Forward_movement,   // "FB_DigIn_16_XOR"
               Input_1 := NOT "HMI_DB".Trolley_movement_mechanism.WP_Forward_movement,
               Input_2 := "HMI_DB".Lifting_mechanism."1YB2_WP_MPP_disconnected_from_brake",
               Input_3 := NOT "HMI_DB".Lifting_mechanism."1YB2_WP_MPP_disconnected_from_brake",
               Input_4 := "HMI_DB".Lifting_mechanism.MD_disconnected_from_drive,
               Input_5 := NOT "HMI_DB".Lifting_mechanism.MD_disconnected_from_drive,
               Input_6 := "HMI_DB".PSM.ID_Line_contactor_from_remote_control_On,
               Input_7 := NOT "HMI_DB".PSM.ID_Line_contactor_from_remote_control_On,
               Input_8 := "HMI_DB".PSM.Line_contactor_On,
               Input_9 := NOT "HMI_DB".PSM.Line_contactor_On,
               Input_10 := "HMI_DB".PSM.Control_contactor_220V_On,
               Input_11 := NOT "HMI_DB".PSM.Control_contactor_220V_On,
               Input_14 := "HMI_DB".PSM.CMD_Line_contactor_enable_permission,
               Input_15 := NOT "HMI_DB".PSM.CMD_Line_contactor_enable_permission,
               ixInit := "xInitMerker",
               owHMI_Word => "HMI_DB".Messages.LinearContactor.wMessageWord4);
END_REGION

REGION Network 7: П'яте слово повідомлень
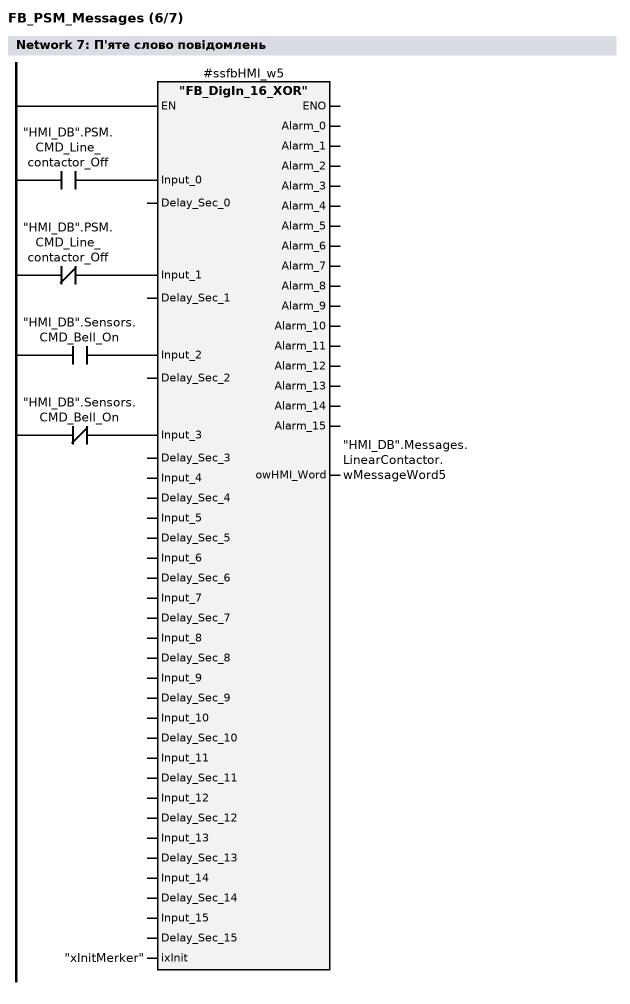
   RUNG wire#powerrail
      #ssfbHMI_w5(Input_0 := wire#w1, Input_1 := wire#w2, Input_2 := wire#w3, Input_3 := wire#w4, Delay_Sec_0 :=, Delay_Sec_1 :=, Delay_Sec_2 :=, Delay_Sec_3 :=, Input_4 :=, Delay_Sec_4 :=, Input_5 :=, Delay_Sec_5 :=, Input_6 :=, Delay_Sec_6 :=, Input_7 :=, Delay_Sec_7 :=, Input_8 :=, Delay_Sec_8 :=, Input_9 :=, Delay_Sec_9 :=, Input_10 :=, Delay_Sec_10 :=, Input_11 :=, Delay_Sec_11 :=, Input_12 :=, Delay_Sec_12 :=, Input_13 :=, Delay_Sec_13 :=, Input_14 :=, Delay_Sec_14 :=, Input_15 :=, Delay_Sec_15 :=, ixInit := "xInitMerker", Alarm_0 =>, Alarm_1 =>, Alarm_2 =>, Alarm_3 =>, Alarm_4 =>, Alarm_5 =>, Alarm_6 =>, Alarm_7 =>, Alarm_8 =>, Alarm_9 =>, Alarm_10 =>, Alarm_11 =>, Alarm_12 =>, Alarm_13 =>, Alarm_14 =>, Alarm_15 =>, owHMI_Word => "HMI_DB".Messages.LinearContactor.wMessageWord5)
   END_RUNG
   RUNG wire#powerrail
      Contact( "HMI_DB".PSM.CMD_Line_contactor_Off )
   END_RUNG wire#w1
   RUNG wire#powerrail
      I_Contact( "HMI_DB".PSM.CMD_Line_contactor_Off )
   END_RUNG wire#w2
   RUNG wire#powerrail
      Contact( "HMI_DB".Sensors.CMD_Bell_On )
   END_RUNG wire#w3
   RUNG wire#powerrail
      I_Contact( "HMI_DB".Sensors.CMD_Bell_On )
   END_RUNG wire#w4
   // the same network as SCL:
   #ssfbHMI_w5(Input_0 := "HMI_DB".PSM.CMD_Line_contactor_Off,   // "FB_DigIn_16_XOR"
               Input_1 := NOT "HMI_DB".PSM.CMD_Line_contactor_Off,
               Input_2 := "HMI_DB".Sensors.CMD_Bell_On,
               Input_3 := NOT "HMI_DB".Sensors.CMD_Bell_On,
               ixInit := "xInitMerker",
               owHMI_Word => "HMI_DB".Messages.LinearContactor.wMessageWord5);
END_REGION

REGION Network 8: Слово повідомлень власні потреби
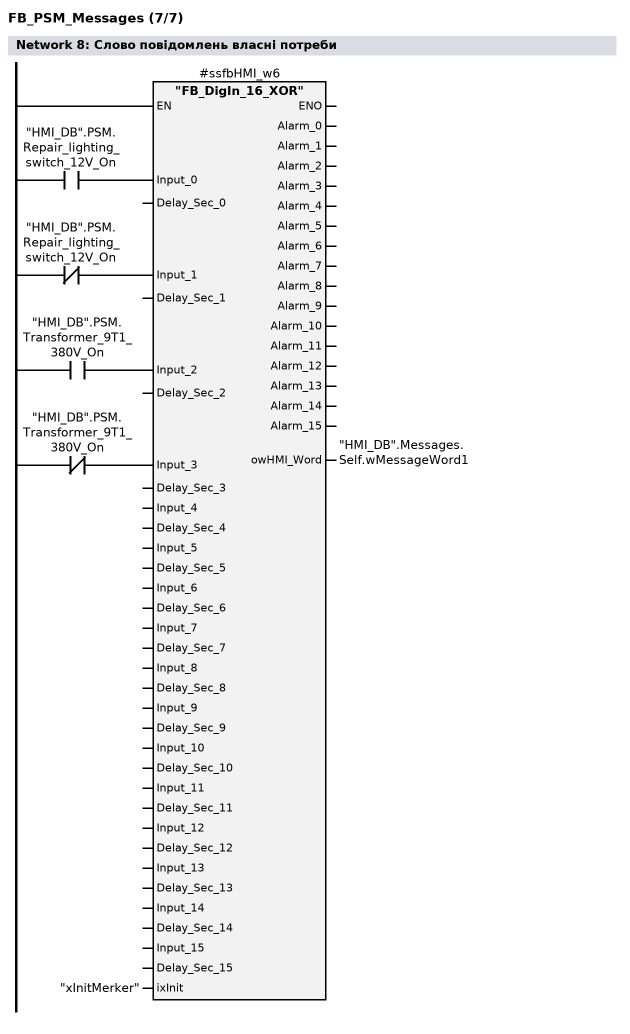
   RUNG wire#powerrail
      #ssfbHMI_w6(Input_0 := wire#w1, Input_1 := wire#w2, Input_2 := wire#w3, Input_3 := wire#w4, Delay_Sec_0 :=, Delay_Sec_1 :=, Delay_Sec_2 :=, Delay_Sec_3 :=, Input_4 :=, Delay_Sec_4 :=, Input_5 :=, Delay_Sec_5 :=, Input_6 :=, Delay_Sec_6 :=, Input_7 :=, Delay_Sec_7 :=, Input_8 :=, Delay_Sec_8 :=, Input_9 :=, Delay_Sec_9 :=, Input_10 :=, Delay_Sec_10 :=, Input_11 :=, Delay_Sec_11 :=, Input_12 :=, Delay_Sec_12 :=, Input_13 :=, Delay_Sec_13 :=, Input_14 :=, Delay_Sec_14 :=, Input_15 :=, Delay_Sec_15 :=, ixInit := "xInitMerker", Alarm_0 =>, Alarm_1 =>, Alarm_2 =>, Alarm_3 =>, Alarm_4 =>, Alarm_5 =>, Alarm_6 =>, Alarm_7 =>, Alarm_8 =>, Alarm_9 =>, Alarm_10 =>, Alarm_11 =>, Alarm_12 =>, Alarm_13 =>, Alarm_14 =>, Alarm_15 =>, owHMI_Word => "HMI_DB".Messages.Self.wMessageWord1)
   END_RUNG
   RUNG wire#powerrail
      Contact( "HMI_DB".PSM.Repair_lighting_switch_12V_On )
   END_RUNG wire#w1
   RUNG wire#powerrail
      I_Contact( "HMI_DB".PSM.Repair_lighting_switch_12V_On )
   END_RUNG wire#w2
   RUNG wire#powerrail
      Contact( "HMI_DB".PSM.Transformer_9T1_380V_On )
   END_RUNG wire#w3
   RUNG wire#powerrail
      I_Contact( "HMI_DB".PSM.Transformer_9T1_380V_On )
   END_RUNG wire#w4
   // the same network as SCL:
   #ssfbHMI_w6(Input_0 := "HMI_DB".PSM.Repair_lighting_switch_12V_On,   // "FB_DigIn_16_XOR"
               Input_1 := NOT "HMI_DB".PSM.Repair_lighting_switch_12V_On,
               Input_2 := "HMI_DB".PSM.Transformer_9T1_380V_On,
               Input_3 := NOT "HMI_DB".PSM.Transformer_9T1_380V_On,
               ixInit := "xInitMerker",
               owHMI_Word => "HMI_DB".Messages.Self.wMessageWord1);
END_REGION
END_FUNCTION_BLOCK

FUNCTION_BLOCK "FB_PSM_Alarms"   // FB22, LAD
{ S7_Optimized_Access := 'TRUE' }
VERSION : 0.1
   VAR
      ssfbAlarmWord1 : "FB_DigIn_16";
      ssfbAlarmWord2 : "FB_DigIn_16";
   END_VAR
BEGIN

REGION Network 2: Перше слово аварій
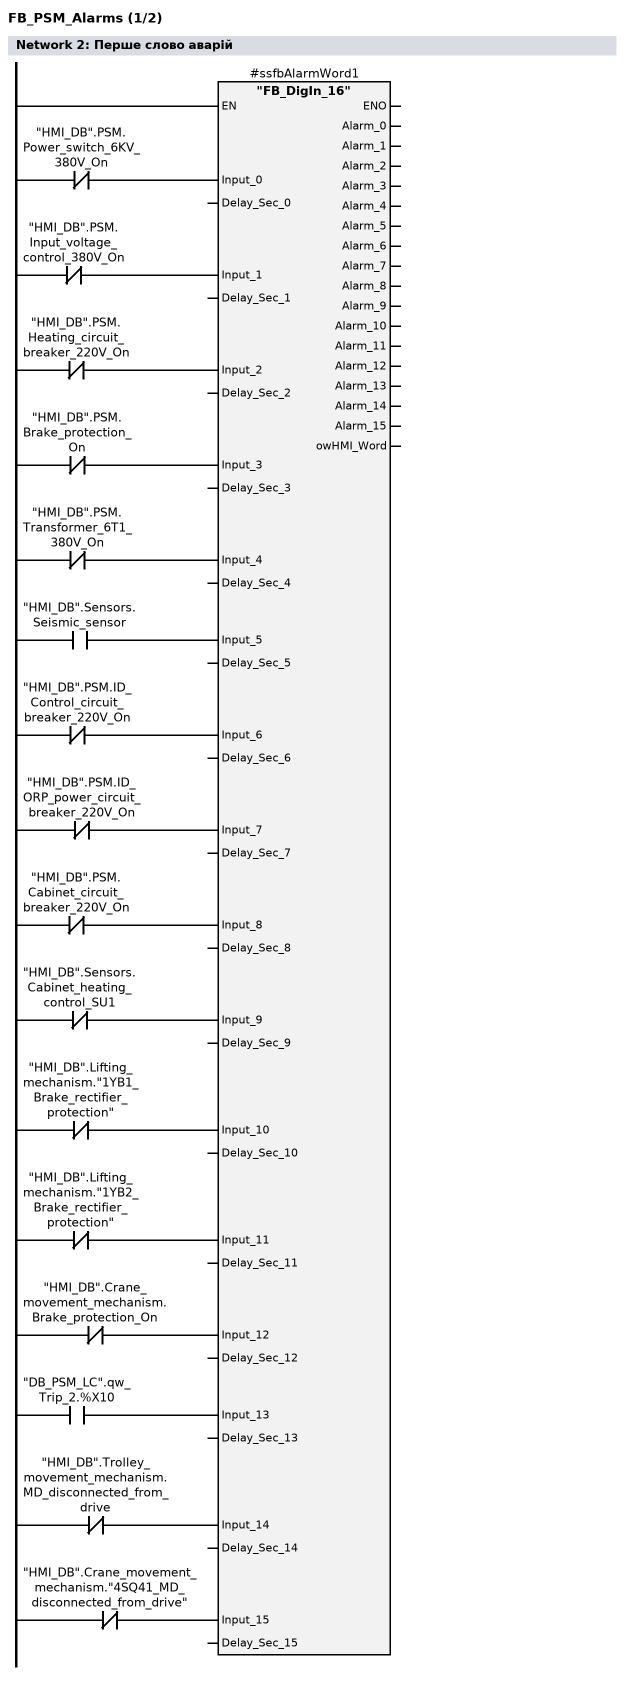
   RUNG wire#powerrail
      #ssfbAlarmWord1(Input_0 := wire#w1, Input_1 := wire#w2, Input_2 := wire#w3, Input_3 := wire#w4, Input_4 := wire#w5, Input_5 := wire#w6, Input_6 := wire#w7, Input_7 := wire#w8, Input_8 := wire#w9, Input_9 := wire#w10, Input_10 := wire#w11, Input_11 := wire#w12, Input_12 := wire#w13, Input_13 := wire#w14, Input_14 := wire#w15, Input_15 := wire#w16, Delay_Sec_0 :=, Delay_Sec_1 :=, Delay_Sec_2 :=, Delay_Sec_3 :=, Delay_Sec_4 :=, Delay_Sec_5 :=, Delay_Sec_6 :=, Delay_Sec_7 :=, Delay_Sec_8 :=, Delay_Sec_9 :=, Delay_Sec_10 :=, Delay_Sec_11 :=, Delay_Sec_12 :=, Delay_Sec_13 :=, Delay_Sec_14 :=, Delay_Sec_15 :=, Alarm_0 =>, Alarm_1 =>, Alarm_2 =>, Alarm_3 =>, Alarm_4 =>, Alarm_5 =>, Alarm_6 =>, Alarm_7 =>, Alarm_8 =>, Alarm_9 =>, Alarm_10 =>, Alarm_11 =>, Alarm_12 =>, Alarm_13 =>, Alarm_14 =>, Alarm_15 =>, owHMI_Word =>)
   END_RUNG
   RUNG wire#powerrail
      I_Contact( "HMI_DB".PSM.Power_switch_6KV_380V_On )
   END_RUNG wire#w1
   RUNG wire#powerrail
      I_Contact( "HMI_DB".PSM.Input_voltage_control_380V_On )
   END_RUNG wire#w2
   RUNG wire#powerrail
      I_Contact( "HMI_DB".PSM.Heating_circuit_breaker_220V_On )
   END_RUNG wire#w3
   RUNG wire#powerrail
      I_Contact( "HMI_DB".PSM.Brake_protection_On )
   END_RUNG wire#w4
   RUNG wire#powerrail
      I_Contact( "HMI_DB".PSM.Transformer_6T1_380V_On )
   END_RUNG wire#w5
   RUNG wire#powerrail
      Contact( "HMI_DB".Sensors.Seismic_sensor )
   END_RUNG wire#w6
   RUNG wire#powerrail
      I_Contact( "HMI_DB".PSM.ID_Control_circuit_breaker_220V_On )
   END_RUNG wire#w7
   RUNG wire#powerrail
      I_Contact( "HMI_DB".PSM.ID_ORP_power_circuit_breaker_220V_On )
   END_RUNG wire#w8
   RUNG wire#powerrail
      I_Contact( "HMI_DB".PSM.Cabinet_circuit_breaker_220V_On )
   END_RUNG wire#w9
   RUNG wire#powerrail
      I_Contact( "HMI_DB".Sensors.Cabinet_heating_control_SU1 )
   END_RUNG wire#w10
   RUNG wire#powerrail
      I_Contact( "HMI_DB".Lifting_mechanism."1YB1_Brake_rectifier_protection" )
   END_RUNG wire#w11
   RUNG wire#powerrail
      I_Contact( "HMI_DB".Lifting_mechanism."1YB2_Brake_rectifier_protection" )
   END_RUNG wire#w12
   RUNG wire#powerrail
      I_Contact( "HMI_DB".Crane_movement_mechanism.Brake_protection_On )
   END_RUNG wire#w13
   RUNG wire#powerrail
      Contact( "DB_PSM_LC".qw_Trip_2.%X10 )
   END_RUNG wire#w14
   RUNG wire#powerrail
      I_Contact( "HMI_DB".Trolley_movement_mechanism.MD_disconnected_from_drive )
   END_RUNG wire#w15
   RUNG wire#powerrail
      I_Contact( "HMI_DB".Crane_movement_mechanism."4SQ41_MD_disconnected_from_drive" )
   END_RUNG wire#w16
   // the same network as SCL:
   #ssfbAlarmWord1(Input_0 := NOT "HMI_DB".PSM.Power_switch_6KV_380V_On,   // "FB_DigIn_16"
                   Input_1 := NOT "HMI_DB".PSM.Input_voltage_control_380V_On,
                   Input_2 := NOT "HMI_DB".PSM.Heating_circuit_breaker_220V_On,
                   Input_3 := NOT "HMI_DB".PSM.Brake_protection_On,
                   Input_4 := NOT "HMI_DB".PSM.Transformer_6T1_380V_On,
                   Input_5 := "HMI_DB".Sensors.Seismic_sensor,
                   Input_6 := NOT "HMI_DB".PSM.ID_Control_circuit_breaker_220V_On,
                   Input_7 := NOT "HMI_DB".PSM.ID_ORP_power_circuit_breaker_220V_On,
                   Input_8 := NOT "HMI_DB".PSM.Cabinet_circuit_breaker_220V_On,
                   Input_9 := NOT "HMI_DB".Sensors.Cabinet_heating_control_SU1,
                   Input_10 := NOT "HMI_DB".Lifting_mechanism."1YB1_Brake_rectifier_protection",
                   Input_11 := NOT "HMI_DB".Lifting_mechanism."1YB2_Brake_rectifier_protection",
                   Input_12 := NOT "HMI_DB".Crane_movement_mechanism.Brake_protection_On,
                   Input_13 := "DB_PSM_LC".qw_Trip_2.%X10,
                   Input_14 := NOT "HMI_DB".Trolley_movement_mechanism.MD_disconnected_from_drive,
                   Input_15 := NOT "HMI_DB".Crane_movement_mechanism."4SQ41_MD_disconnected_from_drive");
END_REGION

REGION Network 3: Друге слово аварій
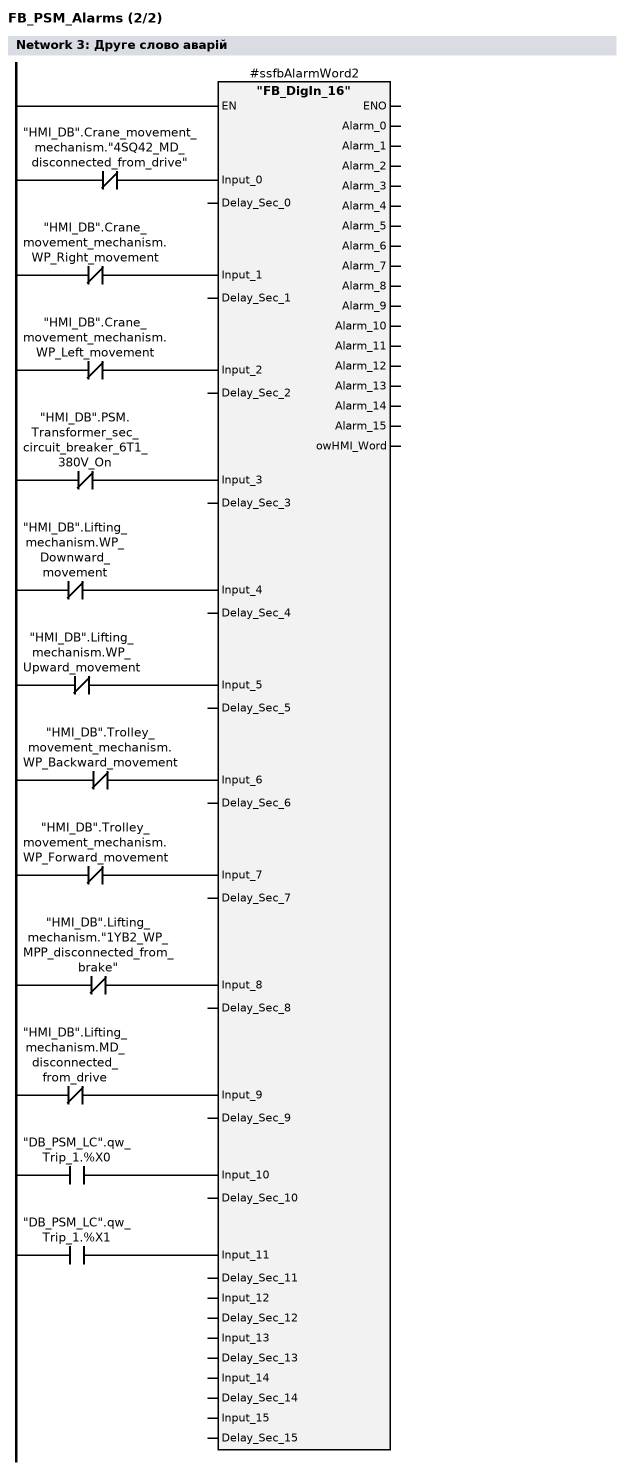
   RUNG wire#powerrail
      #ssfbAlarmWord2(Input_0 := wire#w1, Input_1 := wire#w2, Input_2 := wire#w3, Input_3 := wire#w4, Input_4 := wire#w5, Input_5 := wire#w6, Input_6 := wire#w7, Input_7 := wire#w8, Input_8 := wire#w9, Input_9 := wire#w10, Input_10 := wire#w11, Input_11 := wire#w12, Delay_Sec_0 :=, Delay_Sec_1 :=, Delay_Sec_2 :=, Delay_Sec_3 :=, Delay_Sec_4 :=, Delay_Sec_5 :=, Delay_Sec_6 :=, Delay_Sec_7 :=, Delay_Sec_8 :=, Delay_Sec_9 :=, Delay_Sec_10 :=, Delay_Sec_11 :=, Input_12 :=, Delay_Sec_12 :=, Input_13 :=, Delay_Sec_13 :=, Input_14 :=, Delay_Sec_14 :=, Input_15 :=, Delay_Sec_15 :=, Alarm_0 =>, Alarm_1 =>, Alarm_2 =>, Alarm_3 =>, Alarm_4 =>, Alarm_5 =>, Alarm_6 =>, Alarm_7 =>, Alarm_8 =>, Alarm_9 =>, Alarm_10 =>, Alarm_11 =>, Alarm_12 =>, Alarm_13 =>, Alarm_14 =>, Alarm_15 =>, owHMI_Word =>)
   END_RUNG
   RUNG wire#powerrail
      I_Contact( "HMI_DB".Crane_movement_mechanism."4SQ42_MD_disconnected_from_drive" )
   END_RUNG wire#w1
   RUNG wire#powerrail
      I_Contact( "HMI_DB".Crane_movement_mechanism.WP_Right_movement )
   END_RUNG wire#w2
   RUNG wire#powerrail
      I_Contact( "HMI_DB".Crane_movement_mechanism.WP_Left_movement )
   END_RUNG wire#w3
   RUNG wire#powerrail
      I_Contact( "HMI_DB".PSM.Transformer_sec_circuit_breaker_6T1_380V_On )
   END_RUNG wire#w4
   RUNG wire#powerrail
      I_Contact( "HMI_DB".Lifting_mechanism.WP_Downward_movement )
   END_RUNG wire#w5
   RUNG wire#powerrail
      I_Contact( "HMI_DB".Lifting_mechanism.WP_Upward_movement )
   END_RUNG wire#w6
   RUNG wire#powerrail
      I_Contact( "HMI_DB".Trolley_movement_mechanism.WP_Backward_movement )
   END_RUNG wire#w7
   RUNG wire#powerrail
      I_Contact( "HMI_DB".Trolley_movement_mechanism.WP_Forward_movement )
   END_RUNG wire#w8
   RUNG wire#powerrail
      I_Contact( "HMI_DB".Lifting_mechanism."1YB2_WP_MPP_disconnected_from_brake" )
   END_RUNG wire#w9
   RUNG wire#powerrail
      I_Contact( "HMI_DB".Lifting_mechanism.MD_disconnected_from_drive )
   END_RUNG wire#w10
   RUNG wire#powerrail
      Contact( "DB_PSM_LC".qw_Trip_1.%X0 )
   END_RUNG wire#w11
   RUNG wire#powerrail
      Contact( "DB_PSM_LC".qw_Trip_1.%X1 )
   END_RUNG wire#w12
   // the same network as SCL:
   #ssfbAlarmWord2(Input_0 := NOT "HMI_DB".Crane_movement_mechanism."4SQ42_MD_disconnected_from_drive",   // "FB_DigIn_16"
                   Input_1 := NOT "HMI_DB".Crane_movement_mechanism.WP_Right_movement,
                   Input_2 := NOT "HMI_DB".Crane_movement_mechanism.WP_Left_movement,
                   Input_3 := NOT "HMI_DB".PSM.Transformer_sec_circuit_breaker_6T1_380V_On,
                   Input_4 := NOT "HMI_DB".Lifting_mechanism.WP_Downward_movement,
                   Input_5 := NOT "HMI_DB".Lifting_mechanism.WP_Upward_movement,
                   Input_6 := NOT "HMI_DB".Trolley_movement_mechanism.WP_Backward_movement,
                   Input_7 := NOT "HMI_DB".Trolley_movement_mechanism.WP_Forward_movement,
                   Input_8 := NOT "HMI_DB".Lifting_mechanism."1YB2_WP_MPP_disconnected_from_brake",
                   Input_9 := NOT "HMI_DB".Lifting_mechanism.MD_disconnected_from_drive,
                   Input_10 := "DB_PSM_LC".qw_Trip_1.%X0,
                   Input_11 := "DB_PSM_LC".qw_Trip_1.%X1);
END_REGION
END_FUNCTION_BLOCK

FUNCTION "FC_PSM_General" : Void   // FC20, LAD
{ S7_Optimized_Access := 'TRUE' }
VERSION : 0.1
   VAR_TEMP
      twError : Word;
   END_VAR
BEGIN

REGION Network 2: Лінійний контактор
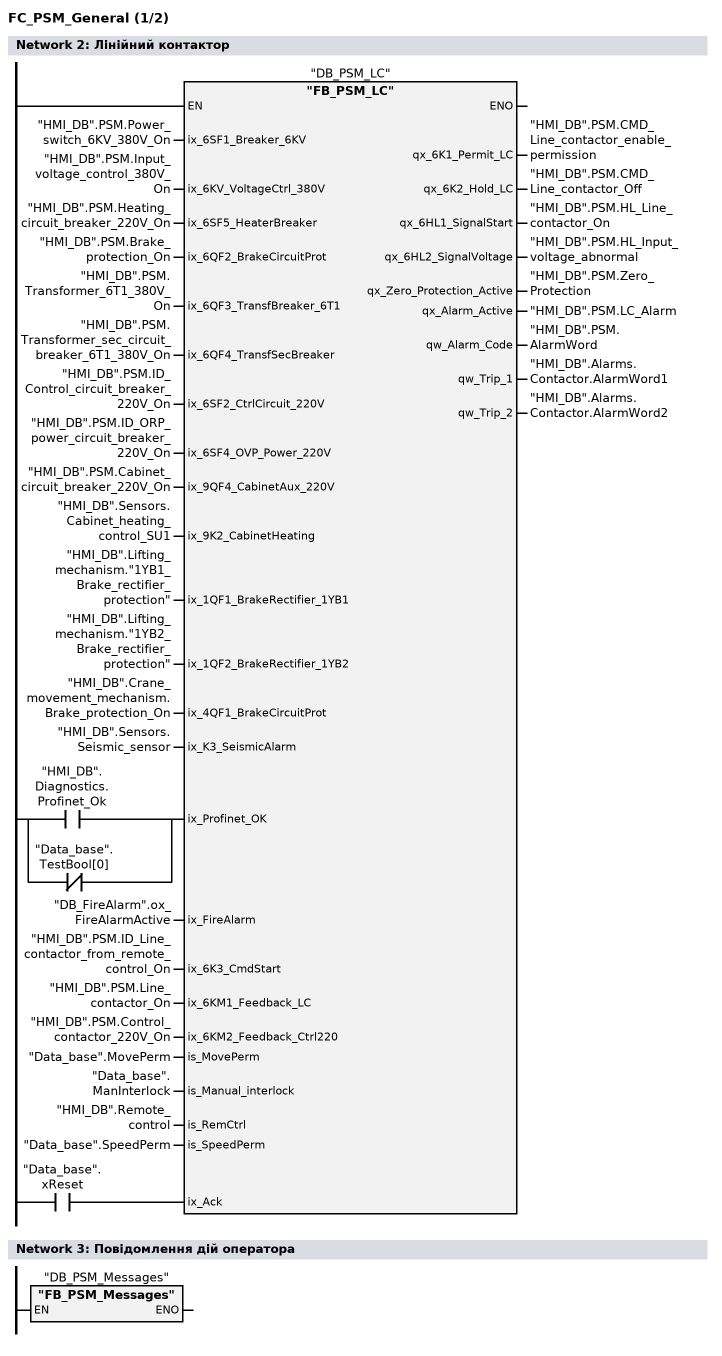
   RUNG wire#powerrail
      "DB_PSM_LC"(ix_Profinet_OK := wire#w1, ix_Ack := wire#w2, ix_6SF1_Breaker_6KV := "HMI_DB".PSM.Power_switch_6KV_380V_On, ix_6KV_VoltageCtrl_380V := "HMI_DB".PSM.Input_voltage_control_380V_On, ix_6SF5_HeaterBreaker := "HMI_DB".PSM.Heating_circuit_breaker_220V_On, ix_6QF2_BrakeCircuitProt := "HMI_DB".PSM.Brake_protection_On, ix_6QF3_TransfBreaker_6T1 := "HMI_DB".PSM.Transformer_6T1_380V_On, ix_6QF4_TransfSecBreaker := "HMI_DB".PSM.Transformer_sec_circuit_breaker_6T1_380V_On, ix_6SF2_CtrlCircuit_220V := "HMI_DB".PSM.ID_Control_circuit_breaker_220V_On, ix_6SF4_OVP_Power_220V := "HMI_DB".PSM.ID_ORP_power_circuit_breaker_220V_On, ix_9QF4_CabinetAux_220V := "HMI_DB".PSM.Cabinet_circuit_breaker_220V_On, ix_9K2_CabinetHeating := "HMI_DB".Sensors.Cabinet_heating_control_SU1, ix_1QF1_BrakeRectifier_1YB1 := "HMI_DB".Lifting_mechanism."1YB1_Brake_rectifier_protection", ix_1QF2_BrakeRectifier_1YB2 := "HMI_DB".Lifting_mechanism."1YB2_Brake_rectifier_protection", ix_4QF1_BrakeCircuitProt := "HMI_DB".Crane_movement_mechanism.Brake_protection_On, ix_K3_SeismicAlarm := "HMI_DB".Sensors.Seismic_sensor, ix_FireAlarm := "DB_FireAlarm".ox_FireAlarmActive, ix_6K3_CmdStart := "HMI_DB".PSM.ID_Line_contactor_from_remote_control_On, ix_6KM1_Feedback_LC := "HMI_DB".PSM.Line_contactor_On, ix_6KM2_Feedback_Ctrl220 := "HMI_DB".PSM.Control_contactor_220V_On, is_MovePerm := "Data_base".MovePerm, is_Manual_interlock := "Data_base".ManInterlock, is_RemCtrl := "HMI_DB".Remote_control, is_SpeedPerm := "Data_base".SpeedPerm, qx_6K1_Permit_LC => "HMI_DB".PSM.CMD_Line_contactor_enable_permission, qx_6K2_Hold_LC => "HMI_DB".PSM.CMD_Line_contactor_Off, qx_6HL1_SignalStart => "HMI_DB".PSM.HL_Line_contactor_On, qx_6HL2_SignalVoltage => "HMI_DB".PSM.HL_Input_voltage_abnormal, qx_Zero_Protection_Active => "HMI_DB".PSM.Zero_Protection, qx_Alarm_Active => "HMI_DB".PSM.LC_Alarm, qw_Alarm_Code => "HMI_DB".PSM.AlarmWord, qw_Trip_1 => "HMI_DB".Alarms.Contactor.AlarmWord1, qw_Trip_2 => "HMI_DB".Alarms.Contactor.AlarmWord2)
   END_RUNG
   RUNG wire#powerrail
      Contact( "HMI_DB".Diagnostics.Profinet_Ok )
   END_RUNG wire#w1
   RUNG wire#powerrail
      I_Contact( "Data_base".TestBool[0] )
   END_RUNG wire#w1
   RUNG wire#powerrail
      Contact( "Data_base".xReset )
   END_RUNG wire#w2
   // the same network as SCL:
   "DB_PSM_LC"(ix_6SF1_Breaker_6KV := "HMI_DB".PSM.Power_switch_6KV_380V_On,   // "FB_PSM_LC"
               ix_6KV_VoltageCtrl_380V := "HMI_DB".PSM.Input_voltage_control_380V_On,
               ix_6SF5_HeaterBreaker := "HMI_DB".PSM.Heating_circuit_breaker_220V_On,
               ix_6QF2_BrakeCircuitProt := "HMI_DB".PSM.Brake_protection_On,
               ix_6QF3_TransfBreaker_6T1 := "HMI_DB".PSM.Transformer_6T1_380V_On,
               ix_6QF4_TransfSecBreaker := "HMI_DB".PSM.Transformer_sec_circuit_breaker_6T1_380V_On,
               ix_6SF2_CtrlCircuit_220V := "HMI_DB".PSM.ID_Control_circuit_breaker_220V_On,
               ix_6SF4_OVP_Power_220V := "HMI_DB".PSM.ID_ORP_power_circuit_breaker_220V_On,
               ix_9QF4_CabinetAux_220V := "HMI_DB".PSM.Cabinet_circuit_breaker_220V_On,
               ix_9K2_CabinetHeating := "HMI_DB".Sensors.Cabinet_heating_control_SU1,
               ix_1QF1_BrakeRectifier_1YB1 := "HMI_DB".Lifting_mechanism."1YB1_Brake_rectifier_protection",
               ix_1QF2_BrakeRectifier_1YB2 := "HMI_DB".Lifting_mechanism."1YB2_Brake_rectifier_protection",
               ix_4QF1_BrakeCircuitProt := "HMI_DB".Crane_movement_mechanism.Brake_protection_On,
               ix_K3_SeismicAlarm := "HMI_DB".Sensors.Seismic_sensor,
               ix_Profinet_OK := "HMI_DB".Diagnostics.Profinet_Ok OR NOT "Data_base".TestBool[0],
               ix_FireAlarm := "DB_FireAlarm".ox_FireAlarmActive,
               ix_6K3_CmdStart := "HMI_DB".PSM.ID_Line_contactor_from_remote_control_On,
               ix_6KM1_Feedback_LC := "HMI_DB".PSM.Line_contactor_On,
               ix_6KM2_Feedback_Ctrl220 := "HMI_DB".PSM.Control_contactor_220V_On,
               is_MovePerm := "Data_base".MovePerm,
               is_Manual_interlock := "Data_base".ManInterlock,
               is_RemCtrl := "HMI_DB".Remote_control,
               is_SpeedPerm := "Data_base".SpeedPerm,
               ix_Ack := "Data_base".xReset,
               qx_6K1_Permit_LC => "HMI_DB".PSM.CMD_Line_contactor_enable_permission,
               qx_6K2_Hold_LC => "HMI_DB".PSM.CMD_Line_contactor_Off,
               qx_6HL1_SignalStart => "HMI_DB".PSM.HL_Line_contactor_On,
               qx_6HL2_SignalVoltage => "HMI_DB".PSM.HL_Input_voltage_abnormal,
               qx_Zero_Protection_Active => "HMI_DB".PSM.Zero_Protection,
               qx_Alarm_Active => "HMI_DB".PSM.LC_Alarm,
               qw_Alarm_Code => "HMI_DB".PSM.AlarmWord,
               qw_Trip_1 => "HMI_DB".Alarms.Contactor.AlarmWord1,
               qw_Trip_2 => "HMI_DB".Alarms.Contactor.AlarmWord2);
END_REGION

REGION Network 3: Повідомлення дій оператора
   RUNG wire#powerrail
      "DB_PSM_Messages"()
   END_RUNG
   // the same network as SCL:
   "DB_PSM_Messages"();   // "FB_PSM_Messages"
END_REGION

REGION Network 4: Аварії
   // Поки що не використуваэмо
END_REGION

REGION Network 5: Підсвічування кнопки
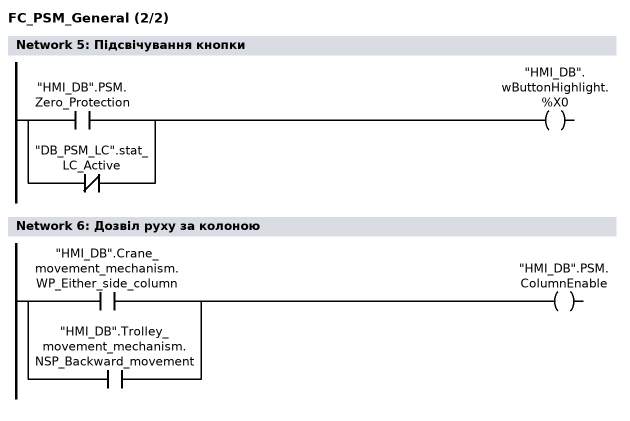
   RUNG wire#powerrail
      Contact( "HMI_DB".PSM.Zero_Protection )
      wire#w1
      Coil( "HMI_DB".wButtonHighlight.%X0 )
   END_RUNG
   RUNG wire#powerrail
      I_Contact( "DB_PSM_LC".stat_LC_Active )
   END_RUNG wire#w1
   // the same network as SCL:
   "HMI_DB".wButtonHighlight.%X0 := "HMI_DB".PSM.Zero_Protection OR NOT "DB_PSM_LC".stat_LC_Active;
END_REGION

REGION Network 6: Дозвіл руху за колоною
   RUNG wire#powerrail
      Contact( "HMI_DB".Crane_movement_mechanism.WP_Either_side_column )
      wire#w1
      Coil( "HMI_DB".PSM.ColumnEnable )
   END_RUNG
   RUNG wire#powerrail
      Contact( "HMI_DB".Trolley_movement_mechanism.NSP_Backward_movement )
   END_RUNG wire#w1
   // the same network as SCL:
   "HMI_DB".PSM.ColumnEnable := "HMI_DB".Crane_movement_mechanism.WP_Either_side_column OR "HMI_DB".Trolley_movement_mechanism.NSP_Backward_movement;
END_REGION
END_FUNCTION

// folder: 300_1UZ1_Lifting(LM)

FUNCTION_BLOCK "FB_Lifting_Control"   // FB300, SCL
{ S7_Optimized_Access := 'TRUE' }
VERSION : 0.1
   VAR_INPUT
      ix_MainContactorON : Bool;   // Головний контактор увімкнено
      Ix_Calibrated : Bool;   // Механізм калібровано
      ix_CalibrationActive : Bool;   // Активна процедура калібровки
      ix_CalibrationBlockUp : Bool;   // Заборона руху вгору від сіквенсера калібровки
      ix_CalibrationBlockDown : Bool;   // Заборона руху вниз від сіквенсера калібровки
      ix_CalibrationQuickStop : Bool;   // Запит Quick Stop від сіквенсера калібровки
      ix_EmergencyStop : Bool;   // Загальний аварійний стоп
      ix_Encoder_RDY : Bool;
      ix_Fault_1UZ1 : Bool;
      ix_1BT1_ThermalResistor : Bool;   // Термостат гальмівного резистора (NC contact, TRUE = Норма)
      ix_1KT_ThermalMotor : Bool;   // Термісторне реле захисту двигуна 1M1 (Аварія = TRUE)
      ix_1BV_DrumRotationCtrl : Bool;   // Перемикач швидкості барабану (NC contact, TRUE = Норма)
      ix_1SQ21_BrakeOpened : Bool;   // Кінцевик «відкрито» (розгальмовано)
      ix_1SQ22_BrakeClosed : Bool;   // Кінцевик «закрито» (загальмовано)
      ix_1SQ23_BrakeLiningsNormal : Bool;   // Кінцевик контролю зносу накладок (TRUE = Норма)
      ix_1BM1_6k_BrakeWearErr : Bool;   // Сигнал діагностичного блоку DUE зносу гальма 1YB1
      is_RemCtrl : "udtRemCtrl";   // Кнопки руху з пульта (для контролю нульового положення при старті)
      is_MovePerm : "udtMovePerm";   // Кінцеві вимикачі руху крайніх положень
      is_SpeedPerm : "udtSpeedPerm";   // Кінцеві вимикачі швидкості руху
      ix_Zone_ProgStopUp : Bool;   // Програмна зона зупинки вгору (по енкодеру)
      ix_Zone_ProgStopDown : Bool;   // Програмна зона зупинки вниз (по енкодеру)
      ix_1K11_Overload115 : Bool;   // Відсутність сигналу = Перевантаження 115%
      ix_1K12_RopeSlack : Bool;   // Відсутність сигналу = Ослаблення канатів / провисання
      ix_1K31_EmergencyBrakeReleased : Bool;   // Аварійне гальмо 1YB2 розгальмоване (кінцевик 1SQ33)
      ix_DriveReleaseBrakeCmd : Bool;   // Команда розгальмування від ЧП 1UZ1 в телеграмі
      ir_Actual_Torque_1A1 : Real;   // Поточний момент з датчика 1А1, Нм
      ir_Drive_Torque_Feedback : Real;   // Поточний момент від ЧП 1UZ1 через Profinet (в Нм)
      ix_Cmd_ResetAlarm : Bool;
   END_VAR
   VAR_OUTPUT
      qx_1KM1_WorkingBrake : Bool;   // Пускач зовнішнього гальма 1MB1
      qx_1KM2_BuiltInBrake : Bool;   // Пускач вбудованого гальма 1YB1
      qx_1KM3_EmergencyBrake : Bool;   // Пускач аварійного гальма 1YB2
      qx_Drive_Enable : Bool;   // Загальний сигнал дозволу руху / роботи ЧП (ON/OFF1)
      qx_Drive_QuickStop : Bool;   // Команда швидкого гальмування Quick Stop (OFF3)
      qr_Drive_SpeedSetpoint : Real;   // Завдання швидкості на ЧП зі знаком (+ вгору, - вниз)
      qx_1HL_Ready : Bool;   // Світловий індикатор готовності підйому (зелений)
      qx_Global_Alarm : Bool;   // Загальний сигнал наявності будь-якої активної аварії
      qw_Alarm_Word : Word;   // Слово аварій для HMI
      Status_Word : Word;   // Слово стану механізму підйому для HMI/Profinet
   END_VAR
   VAR
      EmerBrake_TON : TON_TIME;   // Таймер накладання аварійного гальма (1 хв)
      BrakeTimeout_TON : TON_TIME;   // Таймер контролю датчиків стану гальм
      EmerBrakeTimeout_TON : TON_TIME;
      MotionActive : Bool;   // Ознака активного запиту на рух від оператора
      stat_BlockAfterReset : Bool;   // Прапорець блокування після скидання аварії
      stat_OldGlobalAlarm : Bool;   // Пам'ять попереднього стану аварії для логіки фронтів END_VAR
      Block_Up : Bool;   // Блокування підйому
      Block_Down : Bool;   // Блокування опускання
      statAlarmWord : Word;   // Статичне слово для збереження стану аварій між циклами PLC
   END_VAR
   VAR_TEMP
      GlobalBlock : Bool;   // Загальне блокування руху
      Valid_Cmd_Up : Bool;   // Валідована команда вгору
      Valid_Cmd_Down : Bool;   // Валідована команда вниз
      AtUpperLimit : Bool;   // Тимчасовий прапорець верхнього положення
      AtLowerLimit : Bool;   // Тимчасовий прапорець нижнього положення
      ResetTrigger : Bool;   // Фронт скидання аварії
      tempStatusWord : Word;   // Тимчасова змінна для збірки слова стану
   END_VAR
BEGIN
   // 1. ФОРМУВАННЯ ТА ФІКСАЦІЯ АВАРІЙ У СЛОВІ (LATCH LOGIC)


   // Bit 0: Аварійний стоп
   IF #ix_EmergencyStop THEN
       #statAlarmWord.%X0 := TRUE;
   END_IF;

   // Bit 1: Втрата головного контактора під час роботи
   IF NOT #ix_MainContactorON AND (#MotionActive OR #qx_Drive_Enable) THEN
       #statAlarmWord.%X1 := TRUE;
   END_IF;

   // Bit 2: Перегрів гальмівного резистора (1BT1)
   IF NOT #"ix_1BT1_ThermalResistor" THEN
       #statAlarmWord.%X2 := TRUE;
   END_IF;

   // Bit 3: Перегрів двигуна підйому (1KT)
   IF  NOT #"ix_1KT_ThermalMotor" THEN
       #statAlarmWord.%X3 := TRUE;
   END_IF;

   // Bit 4: Знос колодок робочого гальма (1SQ23)
   IF NOT #"ix_1SQ23_BrakeLiningsNormal" THEN
       #statAlarmWord.%X4 := TRUE;
   END_IF;

   // Bit 5: Знос вбудованого гальма двигуна (1BM1_6k)
   IF NOT #"ix_1BM1_6k_BrakeWearErr" THEN
       #statAlarmWord.%X5 := TRUE;
   END_IF;

   //Bit 6: Контроль обертання барабану (1BV)
   IF NOT #"ix_1BV_DrumRotationCtrl" THEN
       #statAlarmWord.%X6 := TRUE;
   END_IF;

   //#statAlarmWord.%X6 := FALSE;

   // Bit 7: Розбіжність датчика моменту 1А1 та ЧП > 20%
   //IF #MotionActive AND (ABS(#ir_Actual_Torque_1A1 - #ir_Drive_Torque_Feedback) > 20.0) THEN
   //    #statAlarmWord.%X7 := TRUE;
   //END_IF;

   // Bit 8: Перевищення часу розгальмування робочого гальма
   #BrakeTimeout_TON(IN := #"qx_1KM1_WorkingBrake" AND NOT #"ix_1SQ21_BrakeOpened",
                     PT := T#2.5s);
   IF #BrakeTimeout_TON.Q THEN
       #statAlarmWord.%X8 := TRUE;
   END_IF;

   // Bit 9: Несправність частотного перетворювача
   IF #ix_Fault_1UZ1 THEN
       #statAlarmWord.%X9 := TRUE;
   END_IF;

   //Bit 10: Помилка енкодера
   IF NOT #"ix_Encoder_RDY" THEN
       #statAlarmWord.%X10 := TRUE;
   END_IF;

   //Bit 11: Помилка 
   #EmerBrakeTimeout_TON(IN:=(#ix_1SQ21_BrakeOpened AND #ix_1SQ22_BrakeClosed) OR (NOT #ix_1SQ21_BrakeOpened AND NOT #ix_1SQ22_BrakeClosed),
                         PT:=T#2.0s);


   //Bit 12: Помилка

   // Збереження стану загальної аварії перед можливим скиданням
   #stat_OldGlobalAlarm := #statAlarmWord <> 16#0000;

   // 2. СКИДАННЯ АВАРІЙНИХ БІТІВ (КВІТУВАННЯ)
   // Кожен біт очищується лише за умови відсутності фізичної першопричини аварії
   IF #ix_Cmd_ResetAlarm THEN
       IF NOT #ix_EmergencyStop THEN
           #statAlarmWord.%X0 := FALSE;
       END_IF;
       IF #ix_MainContactorON THEN
           #statAlarmWord.%X1 := FALSE;
       END_IF;
       IF #"ix_1BT1_ThermalResistor" THEN
           #statAlarmWord.%X2 := FALSE;
       END_IF;
       IF #"ix_1KT_ThermalMotor" THEN
           #statAlarmWord.%X3 := FALSE;
       END_IF;
       IF #"ix_1SQ23_BrakeLiningsNormal" THEN
           #statAlarmWord.%X4 := FALSE;
       END_IF;
       IF #"ix_1BM1_6k_BrakeWearErr" THEN
           #statAlarmWord.%X5 := FALSE;
       END_IF;
       IF #"ix_1BV_DrumRotationCtrl" THEN
           #statAlarmWord.%X6 := FALSE;
       END_IF;

       // Розрахункові помилки скидаються безумовно
       #statAlarmWord.%X7 := FALSE;
       #statAlarmWord.%X8 := FALSE;

       IF NOT #ix_Fault_1UZ1 THEN
           #statAlarmWord.%X9 := FALSE;
       END_IF;
       IF #"ix_Encoder_RDY" THEN
           #statAlarmWord.%X10 := FALSE;
       END_IF;
   END_IF;

   // Запис сформованого слова на вихід блоку
   #qw_Alarm_Word := #statAlarmWord;
   // Якщо слово не дорівнює нулю (тобто хоча б один біт аварії активний) — видаємо загальний сигнал
   #qx_Global_Alarm := #statAlarmWord <> 16#0000;

   // 3. АВТОМАТИЧНИЙ ЗАХИСТ ВІД ПОВТОРНОГО ПУСКУ (НОВА ЛОГІКА)
   // Визначаємо задній фронт аварії (момент, коли аварія щойно зникла після натискання Reset)
   #ResetTrigger := #stat_OldGlobalAlarm AND NOT #qx_Global_Alarm;

   // Якщо аварію скинули, але оператор продовжує утримувати кнопку ходу вгору чи вниз — активуємо захисне блокування
   IF #ResetTrigger AND (#is_RemCtrl.Btn_Up OR #is_RemCtrl.Btn_Down) OR ((#is_RemCtrl.Btn_Up AND #Block_Up)OR (#is_RemCtrl.Btn_Down AND #Block_Down))THEN
       #stat_BlockAfterReset := TRUE;
   END_IF;

   // Зняття захисного блокування відбувається ТІЛЬКИ тоді, коли пульт переведено в нейтраль (обидві кнопки відпущені)
   IF NOT #is_RemCtrl.Btn_Up AND NOT #is_RemCtrl.Btn_Down THEN
       #stat_BlockAfterReset := FALSE;
   END_IF;

   // 4. ОКРЕМІ ТЕХНОЛОГІЧНІ БЛОКУВАННЯ НАПРЯМКІВ

   //New code 2026-08-10 - O.Husiev
   #Block_Up :=
   NOT #"ix_1K11_Overload115"
   OR NOT #is_MovePerm.Upward
   OR #ix_Zone_ProgStopUp
   OR #ix_CalibrationBlockUp;

   #Block_Down :=
   NOT #"ix_1K12_RopeSlack"
   OR NOT #is_MovePerm.Downward
   OR #ix_Zone_ProgStopDown
   OR #ix_CalibrationBlockDown;


   // 5. ЗАГАЛЬНА ЗАБОРОНА РУХУ (БЛОКУВАННЯ)

   //New code 2026-08-10 - O.Husiev
   #GlobalBlock :=
   #qx_Global_Alarm
   OR NOT #ix_MainContactorON
   OR #stat_BlockAfterReset
   OR (NOT #Ix_Calibrated AND NOT #ix_CalibrationActive)
   OR (#is_RemCtrl.Btn_Up AND #Block_Up)
   OR (#is_RemCtrl.Btn_Down AND #Block_Down);


   // 6. ВАЛІДАЦІЯ КОМАНД ТА АКТИВНІСТЬ РУХУ
   #Valid_Cmd_Up := #is_RemCtrl.Btn_Up AND NOT #GlobalBlock AND NOT #Block_Up; //AND #"ix_1K31_EmergencyBrakeReleased";
   #Valid_Cmd_Down := #is_RemCtrl.Btn_Down AND NOT #GlobalBlock AND NOT #Block_Down; //AND #"ix_1K31_EmergencyBrakeReleased";

   #MotionActive := (#is_RemCtrl.Btn_Up AND NOT #Block_Up) OR (#is_RemCtrl.Btn_Down AND NOT #Block_Down);

   // 7. СВІТЛОВА СИГНАЛІЗАЦІЯ ГОТОВНОСТІ (Зелений індикатор 1HL на пульті)
   #"qx_1HL_Ready" := NOT #GlobalBlock AND #Ix_Calibrated AND #is_MovePerm.Upward AND #is_MovePerm.Downward;

   // 8. КЕРУВАННЯ АВАРІЙНИМ ГАЛЬМОМ (1YB2 через пускач 1KM3)
   #EmerBrake_TON(IN := NOT #MotionActive AND NOT #GlobalBlock,
                  PT := T#1m);

   IF #GlobalBlock THEN
       #"qx_1KM3_EmergencyBrake" := FALSE; // При будь-якій активній аварії — миттєве накладання
   ELSIF #MotionActive THEN
       #"qx_1KM3_EmergencyBrake" := TRUE;
   ELSIF #EmerBrake_TON.Q THEN
       #"qx_1KM3_EmergencyBrake" := FALSE;
   END_IF;

   //#"qx_1KM3_EmergencyBrake" := TRUE;

   // 9. КЕРУВАННЯ РОБОЧИМ ТА ВБУДОВАНИМ ГАЛЬМАМИ (1MB1 -> 1KM1, 1YB1 -> 1KM2)
   IF #ix_DriveReleaseBrakeCmd AND NOT #GlobalBlock THEN
       #"qx_1KM1_WorkingBrake" := TRUE;
       #"qx_1KM2_BuiltInBrake" := TRUE;
   ELSE
       #"qx_1KM1_WorkingBrake" := FALSE;
       #"qx_1KM2_BuiltInBrake" := FALSE;
   END_IF;

   // 10. КЕРУВАННЯ ЧП ЧЕРЕЗ PROFINET
   #qx_Drive_Enable := #ix_1K31_EmergencyBrakeReleased AND (#Valid_Cmd_Up OR #Valid_Cmd_Down);

   // Швидка зупинка Quick Stop (досягнення програмних зон або активна аварія барабану)

   //New code 2026-08-10 - O.Husiev
   #qx_Drive_QuickStop :=
   (#is_RemCtrl.Btn_Up AND #ix_Zone_ProgStopUp)
   OR (#is_RemCtrl.Btn_Down AND #ix_Zone_ProgStopDown)
   OR #statAlarmWord.%X6
   OR #ix_CalibrationQuickStop;


   // ЛОГІКА ЗАДАННЯ ШВИДКОСТІ (+ вгору, - вниз)

   //New code 2026-08-10 - O.Husiev
   IF NOT #qx_Drive_Enable THEN

       #qr_Drive_SpeedSetpoint := 0.0;

   ELSIF #Valid_Cmd_Up THEN

       IF #is_RemCtrl.Btn_ScndSpeed
           AND #is_SpeedPerm.Speed_normal_Up
           AND #"ix_1K12_RopeSlack"
           AND NOT #ix_CalibrationActive
       THEN

           #qr_Drive_SpeedSetpoint := 1000.0;

       ELSE

           #qr_Drive_SpeedSetpoint := 250.0;

       END_IF;

   ELSIF #Valid_Cmd_Down THEN

       IF #is_RemCtrl.Btn_ScndSpeed
           AND #is_SpeedPerm.Speed_normal_Down
           AND NOT #ix_CalibrationActive
       THEN

           #qr_Drive_SpeedSetpoint := -1000.0;

       ELSE

           #qr_Drive_SpeedSetpoint := -250.0;

       END_IF;

   END_IF;


   // 11. ФОРМУВАННЯ ДЕТАЛЬНОГО СЛОВА СТАНУ ПІДЙОМНИКА (Status_Word)
   #tempStatusWord := 16#0000;

   // Допоміжні прапорці досягнення кінцевих точок за ТЗ (фізичний кінцевик або програмна координатна зона)
   #AtUpperLimit := (NOT #is_MovePerm.Upward) OR #ix_Zone_ProgStopUp;
   #AtLowerLimit := (NOT #is_MovePerm.Downward) OR #ix_Zone_ProgStopDown;

   // Оцінка динамічного стану підйомника
   IF #qx_Drive_Enable AND (#qr_Drive_SpeedSetpoint > 0.0) THEN
       #tempStatusWord.%X0 := TRUE;   // Рухається вверх

   ELSIF #qx_Drive_Enable AND (#qr_Drive_SpeedSetpoint < 0.0) THEN
       #tempStatusWord.%X1 := TRUE;   // Рухається вниз

   ELSE
       // АНАЛІЗ СТАНІВ ЗУПИНКИ
       IF #qx_Global_Alarm THEN
           #tempStatusWord.%X4 := TRUE;   // Аварія (найвищий пріоритет зупинки)
       ELSIF #AtUpperLimit THEN
           #tempStatusWord.%X5 := TRUE;   // Зупинено у верхньому положенні
       ELSIF #AtLowerLimit THEN
           #tempStatusWord.%X6 := TRUE;   // Зупинено у нижньому положенні
       ELSIF #qx_1HL_Ready THEN
           #tempStatusWord.%X2 := TRUE;   // Зупинено і Готовий до роботи (в середній зоні)
       ELSE
           #tempStatusWord.%X3 := TRUE;   // Зупинено і НЕ готовий до роботи
       END_IF;
   END_IF;

   // Дублювання біта аварії, якщо вона виникає безпосередньо під час ходу
   IF #qx_Global_Alarm THEN
       #tempStatusWord.%X4 := TRUE;
   END_IF;

   #Status_Word := #tempStatusWord;
END_FUNCTION_BLOCK

FUNCTION_BLOCK "FB_LiftUp_Messages"   // FB321, LAD
{ S7_Optimized_Access := 'TRUE' }
VERSION : 0.1
   VAR
      ssfbHMI_w1 : "FB_DigIn_16_XOR";
      ssfbHMI_w2 : "FB_DigIn_16_XOR";
      ssfbHMI_w3 : "FB_DigIn_16_XOR";
      ssfbHMI_w4 : "FB_DigIn_16_XOR";
      sarrxhmf : Array[0..10] of Bool;
   END_VAR
   VAR_TEMP
      txStartMovement : Bool;   // Початок руху механізма
      txStopMovement : Bool;   // Кінець руху механізма
      twTemp : Word;
   END_VAR
   VAR_TEMP   // added for the SCL form of the ladder/FBD networks
      _w1 : Bool;
      _w2 : Bool;
      _w3 : Bool;
      _w4 : Bool;
   END_VAR
BEGIN

REGION Network 1: Ініціалізація
END_REGION

REGION Network 2 (SCL)

   // початок руху
   #twTemp := "HMI_DB".Lifting_mechanism.LM_Status AND W#16#3;
   #txStartMovement := #twTemp <> 0;
   // кінець руху
   #twTemp := "HMI_DB".Lifting_mechanism.LM_Status AND W#2#01101100;
   #txStopMovement := #twTemp <> 0;
END_REGION

